									ELSE
										Mach_Control.WJ_b.Error[7]:=TRUE;//尾卷下料时卷针旋转不满足下料角度----20240116
									END_IF	
				     END_IF	
			(*	279:
					IF arrAxisCtrl[AxiseNo.AxisName.TailCurlLine].Cmd.arrbRealPoint[4] THEN
						arrAxisCtrl[AxiseNo.AxisName.TailCurlLine].Cmd.iGoSetPos:=0;
							IF Mach_Control.WJ_b.SinStepMode THEN//尾卷单步模式
								TailCurlSinStep:=TRUE;
							ELSE
								TailCurlSinStep:=FALSE;
							END_IF											
									TailCurlStep3:=280;
					ELSE
						arrAxisCtrl[AxiseNo.AxisName.TailCurlLine].Cmd.iGoSetPos:=4;//尾卷夹电芯平移至取电芯位
					END_IF*)
				
				280://尾卷取电芯夹爪气缸平夹紧
						IF NOT TailCurlSinStep THEN				
							arrCyCtrl[arrCyNo.CylinderName.TailCurlSplintCy].Cmd.bON:=TRUE;//尾卷取料夹爪气缸夹紧
							IF arrCyCtrl[arrCyNo.CylinderName.TailCurlSplintCy].Io.DIOnSwitch THEN
								arrCyCtrl[arrCyNo.ElectValveName.WJ_blow].Cmd.bON:=TRUE;//	夹膜电芯吹气开
								IF Mach_Control.WJ_b.SinStepMode THEN//尾卷单步模式
									TailCurlSinStep:=TRUE;
								ELSE
									TailCurlSinStep:=FALSE;
								END_IF	
								TailCurlStep3:=283;
							END_IF
						END_IF
				
				283://夹膜打开
						IF NOT TailCurlSinStep THEN				
							arrCyCtrl[arrCyNo.CylinderName.PoleSplintCy_D].Cmd.bOFF:=TRUE;
							
							IF arrCyCtrl[arrCyNo.CylinderName.PoleSplintCy_D].Status.OFFState THEN
								IF Mach_Control.WJ_b.SinStepMode THEN//尾卷单步模式
									TailCurlSinStep:=TRUE;
								ELSE
									TailCurlSinStep:=FALSE;
								END_IF
								//arrCyCtrl[arrCyNo.ElectValveName.WJ_blow].Cmd.bON:=FALSE;//	夹膜电芯吹气关
								//arrCyCtrl[arrCyNo.ElectValveName.WJ_blow].Cmd.bOFF:=TRUE;//	夹膜电芯吹气关										
								TailCurlStep3:=287;
							END_IF
						END_IF
					
				287:	
					IF arrCyCtrl[arrCyNo.CylinderName.PoleSplintCy_D].Status.OFFState AND NOT arrAxisCtrl[AxiseNo.AxisName.TailCurlSEPTALine].Status.Coupled AND 
							NOT arrAxisCtrl[AxiseNo.AxisName.TailCurlSEPTAUpDown].Status.Coupled THEN
						IF 	 arrAxis[AxiseNo.AxisName.TailCurlSEPTALine].Status.Homed AND arrAxisCtrl[AxiseNo.AxisName.TailCurlSEPTALine].Status.NoMoving THEN
							IF arrAxisCtrl[AxiseNo.AxisName.TailCurlSEPTALine].Cmd.arrbRealPoint[1] THEN
								arrAxisCtrl[AxiseNo.AxisName.TailCurlSEPTALine].Cmd.iGoSetPos:=0;
							ELSE
								arrAxisCtrl[AxiseNo.AxisName.TailCurlSEPTALine].Cmd.iGoSetPos:=1;//尾卷夹隔膜平移初始位
							END_IF
						END_IF	
						IF 	 arrAxisCtrl[AxiseNo.AxisName.TailCurlSEPTAUpDown].Status.Homed AND arrAxisCtrl[AxiseNo.AxisName.TailCurlSEPTAUpDown].Status.NoMoving THEN
							IF arrAxisCtrl[AxiseNo.AxisName.TailCurlSEPTAUpDown].Cmd.arrbRealPoint[1] THEN
								arrAxisCtrl[AxiseNo.AxisName.TailCurlSEPTAUpDown].Cmd.iGoSetPos:=0;
							ELSE
								arrAxisCtrl[AxiseNo.AxisName.TailCurlSEPTAUpDown].Cmd.iGoSetPos:=1;//尾卷夹隔膜升降初始位
							END_IF
						END_IF
						IF 	arrAxisCtrl[AxiseNo.AxisName.TailCurlSEPTALine].Cmd.arrbRealPoint[1] AND  arrAxisCtrl[AxiseNo.AxisName.TailCurlSEPTAUpDown].Cmd.arrbRealPoint[1]  THEN
								IF Mach_Control.WJ_b.SinStepMode THEN//尾卷单步模式
									TailCurlSinStep:=TRUE;
								ELSE
									TailCurlSinStep:=FALSE;
								END_IF				
								TailCurlStep3:=290;	
						END_IF	
					END_IF			








					290://尾卷压轮升降气缸收回、平移气缸收回
						IF NOT TailCurlSinStep THEN		
								arrCyCtrl[arrCyNo.CylinderName.TailCurlUpdownCy].Cmd.bOFF:=TRUE;//尾卷压轮升降气缸收回
								IF arrCyCtrl[arrCyNo.CylinderName.TailCurlUpdownCy].Io.DIOFFSwitch THEN
									arrCyCtrl[arrCyNo.CylinderName.TailCurlLineCy].Cmd.bOFF:=TRUE;//尾卷压轮平移气缸收回		
									IF arrCyCtrl[arrCyNo.CylinderName.TailCurlLineCy].Io.DIOFFSwitch THEN
										IF Mach_Control.WJ_b.SinStepMode THEN//尾卷单步模式
											TailCurlSinStep:=TRUE;
										ELSE
											TailCurlSinStep:=FALSE;
										END_IF	
										TailCurlStep3:=300;
									END_IF
								END_IF
						END_IF
				300://长、短卷针夹电芯气缸泄压、长、短卷针伸缩轴移动至初始位
						IF NOT TailCurlSinStep THEN			
									IF NOT TON_TailCurl[3].Q THEN
										arrCyCtrl[arrCyNo.CylinderName.CurlingSplintCy_L].Cmd.bFree:=TRUE;//尾卷长卷针泄压
										arrCyCtrl[arrCyNo.CylinderName.CurlingSplintCy_S].Cmd.bFree:=TRUE;//尾卷短卷针泄压
										//arrCyCtrl[arrCyNo.ElectValveName.WJShortvacuum].Cmd.bON:=TRUE;//短卷针张开真空开
										//arrCyCtrl[arrCyNo.CylinderName.CurlingSplintCy_S_1].Cmd.bOFF:=TRUE;//尾卷短卷针泄压
										TON_TailCurl[3].IN:=TRUE;
									ELSE
										IF 	arrAxisCtrl[AxiseNo.AxisName.LCurlingneedleLine].Status.Homed AND arrAxisCtrl[AxiseNo.AxisName.LCurlingneedleLine].Status.NoMoving THEN
											IF arrAxisCtrl[AxiseNo.AxisName.LCurlingneedleLine].Cmd.arrbRealPoint[1] THEN
												arrAxisCtrl[AxiseNo.AxisName.LCurlingneedleLine].Cmd.iGoSetPos:=0;
											ELSE
												arrAxisCtrl[AxiseNo.AxisName.LCurlingneedleLine].Cmd.iGoSetPos:=1;
											END_IF
										END_IF
										IF 	arrAxisCtrl[AxiseNo.AxisName.SCurlingneedleLine].Status.Homed AND arrAxisCtrl[AxiseNo.AxisName.SCurlingneedleLine].Status.NoMoving THEN
											IF arrAxisCtrl[AxiseNo.AxisName.SCurlingneedleLine].Cmd.arrbRealPoint[1] THEN
												arrAxisCtrl[AxiseNo.AxisName.SCurlingneedleLine].Cmd.iGoSetPos:=0;
											ELSE
												arrAxisCtrl[AxiseNo.AxisName.SCurlingneedleLine].Cmd.iGoSetPos:=1;
											END_IF
										END_IF
										IF  arrAxisCtrl[AxiseNo.AxisName.LCurlingneedleLine].Cmd.arrbRealPoint[1] AND arrAxisCtrl[AxiseNo.AxisName.SCurlingneedleLine].Cmd.arrbRealPoint[1] THEN
											TON_TailCurl[3].IN:=FALSE;
											arrCyCtrl[arrCyNo.ElectValveName.WJShortvacuum].Cmd.bON:=TRUE;//短卷针张开真空开
											IF Mach_Control.WJ_b.SinStepMode THEN//尾卷单步模式
												TailCurlSinStep:=TRUE;
											ELSE
												TailCurlSinStep:=FALSE;
											END_IF												
											TailCurlStep3:=305;
										END_IF			
									END_IF
							END_IF	
							
				
							
							
							
							
							
							
							
							
							
				310://尾卷夹电芯平移至初始位
						IF NOT TailCurlSinStep THEN				
								IF 	arrCyCtrl[arrCyNo.CylinderName.TailCurlSplintCy].Io.DIOnSwitch AND  arrAxisCtrl[AxiseNo.AxisName.TailCurlLine].Status.Homed AND arrAxisCtrl[AxiseNo.AxisName.TailCurlLine].Status.NoMoving AND
                                         arrAxisCtrl[AxiseNo.AxisName.LCurlingneedleLine].Cmd.arrbRealPoint[1]  AND arrAxisCtrl[AxiseNo.AxisName.SCurlingneedleLine].Cmd.arrbRealPoint[1]  THEN
									IF arrAxisCtrl[AxiseNo.AxisName.TailCurlLine].Cmd.arrbRealPoint[1] THEN
										arrAxisCtrl[AxiseNo.AxisName.TailCurlLine].Cmd.iGoSetPos:=0;
											IF Mach_Control.WJ_b.SinStepMode THEN//尾卷单步模式
												TailCurlSinStep:=TRUE;
											ELSE
												TailCurlSinStep:=FALSE;
											END_IF										
										TailCurlStep3:=315;
									ELSE
										arrAxisCtrl[AxiseNo.AxisName.TailCurlLine].Cmd.iGoSetPos:=1;//尾卷夹电芯平移至初始位
									END_IF
								END_IF
						END_IF
				
					
						
						315://尾卷夹电芯升降至下电芯位      
						  IF NOT TailCurlSinStep THEN		                                                                                                                                                                                                                                                                                                                                                                                                   		
									IF arrAxisCtrl[AxiseNo.AxisName.TailCurlUpDown].Status.Homed AND arrAxisCtrl[AxiseNo.AxisName.TailCurlUpDown].Status.NoMoving THEN
										IF arrAxisCtrl[AxiseNo.AxisName.TailCurlUpDown].Cmd.arrbRealPoint[3] THEN
											arrAxisCtrl[AxiseNo.AxisName.TailCurlUpDown].Cmd.iGoSetPos:=0;
											IF Mach_Control.WJ_b.SinStepMode THEN//尾卷单步模式
												TailCurlSinStep:=TRUE;
											ELSE
												TailCurlSinStep:=FALSE;
											END_IF									
											TailCurlStep3:=320;
										ELSE
											arrAxisCtrl[AxiseNo.AxisName.TailCurlUpDown].Cmd.iGoSetPos:=3;//尾卷夹电芯升降至下电芯位
										END_IF
									END_IF
							END_IF	
						
						
						
						
				320://尾卷夹电芯旋转至下电芯位
						IF NOT TailCurlSinStep THEN				
								IF 	arrCyCtrl[arrCyNo.CylinderName.TailCurlSplintCy].Status.ONState AND  arrAxisCtrl[AxiseNo.AxisName.TailCurlLine].Status.Homed 
									AND arrAxisCtrl[AxiseNo.AxisName.TailCurlLine].Status.NoMoving AND arrAxisCtrl[AxiseNo.AxisName.GluingLine].Status.Homed AND
									arrAxisCtrl[AxiseNo.AxisName.GluingLine].Status.fActPos<=arrAxispar[AxiseNo.AxisName.GluingLine].arrTargetPoint[10] 
									AND NOT Mach_Control.TJ_b.StickerFlag  THEN
									IF arrAxisCtrl[AxiseNo.AxisName.TailCurlWhirling].Cmd.arrbRealPoint[2] THEN
										arrAxisCtrl[AxiseNo.AxisName.TailCurlWhirling].Cmd.iGoSetPos:=0;
											IF Mach_Control.WJ_b.SinStepMode THEN//尾卷单步模式
												TailCurlSinStep:=TRUE;
											ELSE
												TailCurlSinStep:=FALSE;
											END_IF										
										TailCurlStep3:=325;
									ELSE
										arrAxisCtrl[AxiseNo.AxisName.TailCurlWhirling].Cmd.iGoSetPos:=2;//尾卷夹电芯平移至下电芯位
									END_IF
								END_IF
						END_IF		
						
				
						
			
				325:
				//尾卷夹电芯去避让位   
					(*	  IF NOT TailCurlSinStep THEN		                                                                                                                                                                                                                                                                                                                                                                                                   		
									IF arrAxisCtrl[AxiseNo.AxisName.TailCurlLine].Status.Homed AND arrAxisCtrl[AxiseNo.AxisName.TailCurlLine].Status.NoMoving THEN
										IF arrAxisCtrl[AxiseNo.AxisName.TailCurlLine].Cmd.arrbRealPoint[5] THEN
											arrAxisCtrl[AxiseNo.AxisName.TailCurlLine].Cmd.iGoSetPos:=0;
											IF Mach_Control.WJ_b.SinStepMode THEN//尾卷单步模式
												TailCurlSinStep:=TRUE;
											ELSE
												TailCurlSinStep:=FALSE;
											END_IF									
											TailCurlStep3:=330;
										ELSE
											arrAxisCtrl[AxiseNo.AxisName.TailCurlLine].Cmd.iGoSetPos:=5;//尾卷夹电芯平移至避让位
										END_IF
									END_IF
							END_IF*)
				//尾卷夹电芯去下料避让位
							IF NOT TailCurlSinStep THEN		                                                                                                                                                                                                                                                                                                                                                                                                   		
									IF arrAxisCtrl[AxiseNo.AxisName.TailCurlLine].Status.Homed AND arrAxisCtrl[AxiseNo.AxisName.TailCurlLine].Status.NoMoving THEN
										IF arrAxisCtrl[AxiseNo.AxisName.TailCurlLine].Cmd.arrbRealPoint[10] THEN
											arrAxisCtrl[AxiseNo.AxisName.TailCurlLine].Cmd.iGoSetPos:=0;
											IF Mach_Control.WJ_b.SinStepMode THEN//尾卷单步模式
												TailCurlSinStep:=TRUE;
											ELSE
												TailCurlSinStep:=FALSE;
											END_IF									
											TailCurlStep3:=330;
										ELSE
											arrAxisCtrl[AxiseNo.AxisName.TailCurlLine].Cmd.iGoSetPos:=10;//尾卷夹电芯平移至避让位
										END_IF
									END_IF
							END_IF
				330:
						IF NOT TailCurlSinStep THEN
								Mach_Control.WJ_b.TailCultOffloading:=TRUE;//下电芯请求														
								TailCurlStep3:=332;
								
								IF Mach_Control.WJ_b.SinStepMode THEN//尾卷单步模式
									TailCurlSinStep:=TRUE;
								ELSE
									TailCurlSinStep:=FALSE;
								END_IF					
						END_IF				
						

				332:   ///////////////////
						
					IF 	arrAxisCtrl[AxiseNo.AxisName.GluingLine].Cmd.arrbRealPoint[8] AND arrAxisCtrl[AxiseNo.AxisName.GluingLine].Status.NoMoving
						AND arrAxisCtrl[AxiseNo.AxisName.GluingWhirling].Cmd.arrbRealPoint[5] AND arrAxisCtrl[AxiseNo.AxisName.GluingWhirling].Status.NoMoving
						AND arrCyCtrl[arrCyNo.CylinderName.PullGlueModelCy].Status.ONState AND NOT arrCyCtrl[arrCyNo.CylinderName.PullGlueModelCy].Status.Error2 
						AND arrAxisCtrl[AxiseNo.AxisName.TailCurlLine].Status.Homed AND arrAxisCtrl[AxiseNo.AxisName.TailCurlLine].Status.NoMoving	
						AND NOT Mach_Control.TJ_b.StickerDone  AND NOT Mach_Control.TJ_b.StickerFlag
						AND NOT CellMemory[Mach_Control.TJ_b.TJ_Memory].Cell AND NOT Mach_Control.se.GluebHave	THEN
						TailCurlStep3:=335;

					END_IF
						
				335:
						IF arrAxisCtrl[AxiseNo.AxisName.TailCurlLine].Cmd.arrbRealPoint[6] THEN
							arrAxisCtrl[AxiseNo.AxisName.TailCurlLine].Cmd.iGoSetPos:=0;
							IF Mach_Control.WJ_b.SinStepMode THEN//尾卷单步模式
								TailCurlSinStep:=TRUE;
							ELSE
								TailCurlSinStep:=FALSE;
							END_IF									
							TailCurlStep3:=336;
						ELSE
							arrAxisCtrl[AxiseNo.AxisName.TailCurlLine].Cmd.iGoSetPos:=6;//尾卷夹电芯平移至下电芯位
						END_IF
						
				336:
							IF NOT TailCurlSinStep THEN		
									IF 	arrAxisCtrl[AxiseNo.AxisName.GluingLine].Cmd.arrbRealPoint[8] AND arrAxisCtrl[AxiseNo.AxisName.GluingLine].Status.NoMoving
										AND arrAxisCtrl[AxiseNo.AxisName.GluingWhirling].Cmd.arrbRealPoint[5] AND arrAxisCtrl[AxiseNo.AxisName.GluingWhirling].Status.NoMoving
										AND arrCyCtrl[arrCyNo.CylinderName.PullGlueModelCy].Status.ONState AND NOT arrCyCtrl[arrCyNo.CylinderName.PullGlueModelCy].Status.Error2 
										AND arrAxisCtrl[AxiseNo.AxisName.TailCurlRetracting].Status.Homed AND arrAxisCtrl[AxiseNo.AxisName.TailCurlRetracting].Status.NoMoving		THEN
									IF arrAxisCtrl[AxiseNo.AxisName.TailCurlRetracting].Cmd.arrbRealPoint[3] THEN
										arrAxisCtrl[AxiseNo.AxisName.TailCurlRetracting].Cmd.iGoSetPos:=0;
										IF Mach_Control.WJ_b.SinStepMode THEN//尾卷单步模式
											TailCurlSinStep:=TRUE;
										ELSE
											TailCurlSinStep:=FALSE;
										END_IF									
										TailCurlStep3:=337;
									ELSE
										arrAxisCtrl[AxiseNo.AxisName.TailCurlRetracting].Cmd.iGoSetPos:=3;//尾卷夹电芯伸缩至下电芯位
										END_IF
									END_IF
							END_IF	
				337:
							IF NOT TailCurlSinStep THEN			
								IF 	arrAxisCtrl[AxiseNo.AxisName.TailCurlUpDown].Status.Homed AND arrAxisCtrl[AxiseNo.AxisName.TailCurlUpDown].Status.NoMoving  THEN
									IF arrAxisCtrl[AxiseNo.AxisName.TailCurlUpDown].Cmd.arrbRealPoint[4] THEN
													arrAxisCtrl[AxiseNo.AxisName.TailCurlUpDown].Cmd.iGoSetPos:=0;
													IF Mach_Control.WJ_b.SinStepMode THEN//尾卷单步模式
													TailCurlSinStep:=TRUE;
													ELSE
														TailCurlSinStep:=FALSE;
													END_IF	
													TailCurlStep3:=338;
									ELSE
													arrAxisCtrl[AxiseNo.AxisName.TailCurlUpDown].Cmd.iGoSetPos:=4;//尾卷夹电芯升降至下电芯位
									END_IF
								END_IF	
						END_IF				
						
						
						
						
						
						
				338:
				
						IF NOT TailCurlSinStep THEN				
							arrCyCtrl[arrCyNo.CylinderName.PullGlueModelCy].Cmd.bOFF:=TRUE;//贴胶治具气缸闭合
							IF arrCyCtrl[arrCyNo.CylinderName.PullGlueModelCy].Status.OFFState THEN
								IF Mach_Control.WJ_b.SinStepMode THEN//尾卷单步模式
									TailCurlSinStep:=TRUE;
								ELSE
									TailCurlSinStep:=FALSE;
								END_IF										
								TailCurlStep3:=339;
							END_IF
						END_IF


				339:
				

					IF NOT TailCurlSinStep THEN				
							arrCyCtrl[arrCyNo.CylinderName.TailCurlSplintCy].Cmd.bOFF:=TRUE;//尾卷夹爪气缸打开
							IF arrCyCtrl[arrCyNo.CylinderName.TailCurlSplintCy].Status.OFFState THEN
								arrCyCtrl[arrCyNo.ElectValveName.WJ_blow].Cmd.bOFF:=TRUE;//	夹膜电芯吹气关
								IF Mach_Control.WJ_b.SinStepMode THEN//尾卷单步模式
									TailCurlSinStep:=TRUE;
								ELSE
									TailCurlSinStep:=FALSE;
								END_IF	
								Mach_Control.TJ_b.StickerFlag:=TRUE;//置位贴胶夹爪有料标记
								TailCurlStep3:=340;
							END_IF
						END_IF

				340:
					IF NOT TailCurlSinStep THEN			
						IF 	arrAxisCtrl[AxiseNo.AxisName.TailCurlUpDown].Status.Homed AND arrAxisCtrl[AxiseNo.AxisName.TailCurlUpDown].Status.NoMoving  AND
							arrAxisCtrl[AxiseNo.AxisName.TailCurlUpDown].Cmd.arrbRealPoint[4] THEN
							arrAxisPar[AxiseNo.AxisName.TailCurlUpDown].fVelocity_of_Rel := 20   ;
							arrAxisCtrl[AxiseNo.AxisName.TailCurlUpDown].Cmd.fPosition_of_Rel :=3 ;
							arrAxisCtrl[AxiseNo.AxisName.TailCurlUpDown].Cmd.bMoveRel :=  TRUE ;
						END_IF
							IF arrAxis[AxiseNo.AxisName.TailCurlUpDown].NcToPlc.SetPos-arrAxisPar[AxiseNo.AxisName.TailCurlUpDown].arrTargetPoint[4] >=3  
							AND arrAxisCtrl[AxiseNo.AxisName.TailCurlUpDown].Status.NoMoving THEN
								IF Mach_Control.WJ_b.SinStepMode THEN//尾卷单步模式
									TailCurlSinStep:=TRUE;
								ELSE
									TailCurlSinStep:=FALSE;
								END_IF
								TailCurlStep3:=341;
							END_IF
					END_IF	
							
				341:// 尾卷夹电芯平移至避让位

						IF NOT TailCurlSinStep THEN			
								IF 	arrAxisCtrl[AxiseNo.AxisName.TailCurlLine].Status.Homed AND arrAxisCtrl[AxiseNo.AxisName.TailCurlLine].Status.NoMoving THEN
									IF arrAxisCtrl[AxiseNo.AxisName.TailCurlLine].Cmd.arrbRealPoint[10] THEN
										arrAxisCtrl[AxiseNo.AxisName.TailCurlLine].Cmd.iGoSetPos:=0;
									IF Mach_Control.WJ_b.SinStepMode THEN//尾卷单步模式
									TailCurlSinStep:=TRUE;
								ELSE
									TailCurlSinStep:=FALSE;
								END_IF	
										TailCurlStep3:=343;
									ELSE
										arrAxisCtrl[AxiseNo.AxisName.TailCurlLine].Cmd.iGoSetPos:=10;//尾卷夹电芯平移至避让位
									END_IF
								END_IF	
						END_IF	
				343:	
					CellMemory[Mach_Control.TJ_b.TJ_Memory]:=CellMemory[Mach_Control.WJ_b.WJ_Memory];
					MEMSET(ADR(CellMemory[Mach_Control.WJ_b.WJ_Memory]),0,SIZEOF(CellMemory[Mach_Control.WJ_b.WJ_Memory]));		
					TailCurlStep3:=345;		
						
						
						
						
						
						
						
				345:
		
						IF NOT TailCurlSinStep THEN			
								IF 	arrAxisCtrl[AxiseNo.AxisName.TailCurlRetracting].Status.Homed AND arrAxisCtrl[AxiseNo.AxisName.TailCurlRetracting].Status.NoMoving THEN
									IF arrAxisCtrl[AxiseNo.AxisName.TailCurlRetracting].Cmd.arrbRealPoint[1] THEN
										arrAxisCtrl[AxiseNo.AxisName.TailCurlRetracting].Cmd.iGoSetPos:=0;
										IF Mach_Control.WJ_b.SinStepMode THEN//尾卷单步模式
									TailCurlSinStep:=TRUE;
								ELSE
									TailCurlSinStep:=FALSE;
								END_IF	
										
										TailCurlStep3:=350;
									ELSE
										arrAxisCtrl[AxiseNo.AxisName.TailCurlRetracting].Cmd.iGoSetPos:=1;//尾卷夹电芯伸缩回到初始位
									END_IF
								END_IF	
						END_IF	
						
						
						
						
				350:
				IF NOT TailCurlSinStep THEN		
					 IF arrAxisCtrl[AxiseNo.AxisName.GluingLine].Status.fActPos<=arrAxispar[AxiseNo.AxisName.GluingLine].arrTargetPoint[10] 
						AND arrAxisCtrl[AxiseNo.AxisName.GluingLine].Status.Homed AND NOT Mach_Control.WJ_b.TailCultOffloading AND arrAxisCtrl[AxiseNo.AxisName.TailCurlLine].Status.Homed 
						AND arrAxisCtrl[AxiseNo.AxisName.TailCurlLine].Status.NoMoving THEN
						
								IF arrAxisCtrl[AxiseNo.AxisName.TailCurlLine].Cmd.arrbRealPoint[1] THEN
									IF Mach_Control.WJ_b.SinStepMode THEN//尾卷单步模式
									TailCurlSinStep:=TRUE;
								ELSE
									TailCurlSinStep:=FALSE;
								END_IF	
									arrAxisCtrl[AxiseNo.AxisName.TailCurlLine].Cmd.iGoSetPos:=0;
									
									TailCurlStep3:=355;
								ELSE
									arrAxisCtrl[AxiseNo.AxisName.TailCurlLine].Cmd.iGoSetPos:=1;//尾卷夹电芯平移至初始位
								END_IF
						END_IF	
				END_IF	

				355:
							IF NOT TailCurlSinStep THEN			
								IF 	arrAxisCtrl[AxiseNo.AxisName.TailCurlUpDown].Status.Homed AND arrAxisCtrl[AxiseNo.AxisName.TailCurlUpDown].Status.NoMoving  THEN
									IF arrAxisCtrl[AxiseNo.AxisName.TailCurlUpDown].Cmd.arrbRealPoint[4] THEN
													arrAxisCtrl[AxiseNo.AxisName.TailCurlUpDown].Cmd.iGoSetPos:=0;
													IF Mach_Control.WJ_b.SinStepMode THEN//尾卷单步模式
													TailCurlSinStep:=TRUE;
													ELSE
														TailCurlSinStep:=FALSE;
													END_IF	
													TailCurlStep3:=360;
									ELSE
													arrAxisCtrl[AxiseNo.AxisName.TailCurlUpDown].Cmd.iGoSetPos:=4;//尾卷夹电芯升降至下电芯位
									END_IF
								END_IF	
						END_IF
				360:
					IF NOT TailCurlSinStep THEN		
					 IF arrAxisCtrl[AxiseNo.AxisName.GluingLine].Status.fActPos<=arrAxispar[AxiseNo.AxisName.GluingLine].arrTargetPoint[10] 
						AND arrAxisCtrl[AxiseNo.AxisName.GluingLine].Status.Homed AND NOT Mach_Control.WJ_b.TailCultOffloading AND arrAxis[AxiseNo.AxisName.TailCurlWhirling].Status.Homed 
						AND arrAxisCtrl[AxiseNo.AxisName.TailCurlWhirling].Status.NoMoving AND arrAxisCtrl[AxiseNo.AxisName.TailCurlLine].Status.NoMoving AND arrAxisCtrl[AxiseNo.AxisName.TailCurlLine].Cmd.arrbRealPoint[1] THEN
						
								IF arrAxisCtrl[AxiseNo.AxisName.TailCurlWhirling].Cmd.arrbRealPoint[1] THEN
									IF Mach_Control.WJ_b.SinStepMode THEN//尾卷单步模式
									TailCurlSinStep:=TRUE;
								ELSE
									TailCurlSinStep:=FALSE;
								END_IF	
									arrAxisCtrl[AxiseNo.AxisName.TailCurlWhirling].Cmd.iGoSetPos:=0;
									//Mach_Control.WJ_b.TailCultOffloadingDone:=TRUE;
									TailCurlStep3:=370;
								ELSE
									arrAxisCtrl[AxiseNo.AxisName.TailCurlWhirling].Cmd.iGoSetPos:=1;//尾卷夹电芯旋转至取电芯位
								END_IF
						END_IF	
				END_IF	
                
				 370://尾卷夹电芯平移去取电芯等待位
					 IF NOT TailCurlSinStep THEN	
							 IF  arrAxisCtrl[AxiseNo.AxisName.TailCurlUpDown].Status.Homed AND arrAxisCtrl[AxiseNo.AxisName.TailCurlUpDown].Status.NoMoving THEN
											IF arrAxisCtrl[AxiseNo.AxisName.TailCurlUpDown].Cmd.arrbRealPoint[1] THEN
												arrAxisCtrl[AxiseNo.AxisName.TailCurlUpDown].Cmd.iGoSetPos:=0;
											ELSE
												arrAxisCtrl[AxiseNo.AxisName.TailCurlUpDown].Cmd.iGoSetPos:=1;//尾卷夹升降去取电芯高度
											END_IF
							 END_IF
						 
						   IF arrAxisCtrl[AxiseNo.AxisName.TailCurlWhirling].Cmd.arrbRealPoint[1] AND arrAxisCtrl[AxiseNo.AxisName.TailCurlUpDown].Cmd.arrbRealPoint[1] AND
							  arrAxisCtrl[AxiseNo.AxisName.TailCurlSEPTALine].Cmd.arrbRealPoint[1] AND  arrAxisCtrl[AxiseNo.AxisName.TailCurlSEPTAUpDown].Cmd.arrbRealPoint[1] AND
							  arrAxisCtrl[AxiseNo.AxisName.LCurlingneedleLine].Cmd.arrbRealPoint[1] AND arrAxisCtrl[AxiseNo.AxisName.SCurlingneedleLine].Cmd.arrbRealPoint[1] AND
							  arrCyCtrl[arrCyNo.CylinderName.PoleSplintCy_D].Io.DIOFFSwitch AND arrCyCtrl[arrCyNo.CylinderName.TailCurlUpdownCy].Io.DIOFFSwitch AND
							  arrAxisCtrl[AxiseNo.AxisName.TailCurlLine].Status.Homed AND arrAxisCtrl[AxiseNo.AxisName.TailCurlLine].Status.NoMoving  THEN
								   IF arrAxisCtrl[AxiseNo.AxisName.TailCurlLine].Cmd.arrbRealPoint[11]  THEN
									  arrAxisCtrl[AxiseNo.AxisName.TailCurlLine].Cmd.iGoSetPos:=0;
										IF Mach_Control.WJ_b.SinStepMode THEN//尾卷单步模式
										   TailCurlSinStep:=TRUE;
										ELSE
										   TailCurlSinStep:=FALSE;
										END_IF									
										   TailCurlStep3:=0;
										   TailCurlTorMark:=FALSE;//尾卷夹电芯平移力矩判断标志位
								   ELSE
									   arrAxisCtrl[AxiseNo.AxisName.TailCurlLine].Cmd.iGoSetPos:=11;//尾卷夹电芯平移去取电芯等待位
									   TailCurlTorMark:=TRUE;//尾卷夹电芯平移力矩判断标志位
								   END_IF   
							END_IF
						END_IF
				//////////////////////////////////////////////////////////////////////////////////////
				///////////////////////////////////叠台空叠隔膜不尾卷/////////////////////////////////////////////////////
				900:
					    IF NOT TailCurlSinStep THEN
							IF  Mach_Control.DT_b.OffloadRequest AND DP_Step0=6040  THEN
								IF 	arrAxisCtrl[AxiseNo.AxisName.TailCurlUpDown].Status.Homed AND arrAxisCtrl[AxiseNo.AxisName.TailCurlUpDown].Status.NoMoving THEN
										IF arrAxisCtrl[AxiseNo.AxisName.TailCurlUpDown].Cmd.arrbRealPoint[1] THEN//尾卷夹电芯升降初始位
											arrAxisCtrl[AxiseNo.AxisName.TailCurlUpDown].Cmd.iGoSetPos:=0;
										ELSE
											arrAxisCtrl[AxiseNo.AxisName.TailCurlUpDown].Cmd.iGoSetPos:=1;
										END_IF
									END_IF	
								IF 	arrAxisCtrl[AxiseNo.AxisName.TailCurlSEPTAUpDown].Status.Homed AND arrAxisCtrl[AxiseNo.AxisName.TailCurlSEPTAUpDown].Status.NoMoving THEN
										IF arrAxisCtrl[AxiseNo.AxisName.TailCurlSEPTAUpDown].Cmd.arrbRealPoint[1] THEN//夹膜升降初始位
											arrAxisCtrl[AxiseNo.AxisName.TailCurlSEPTAUpDown].Cmd.iGoSetPos:=0;
										ELSE
											arrAxisCtrl[AxiseNo.AxisName.TailCurlSEPTAUpDown].Cmd.iGoSetPos:=1;
										END_IF
									END_IF	
									IF 	arrAxisCtrl[AxiseNo.AxisName.TailCurlUpDown].Cmd.arrbRealPoint[1]  AND arrAxisCtrl[AxiseNo.AxisName.TailCurlUpDown].Cmd.arrbRealPoint[1] 
										AND arrAxisCtrl[AxiseNo.AxisName.TailCurlSEPTAUpDown].Cmd.arrbRealPoint[1]  AND arrAxisCtrl[AxiseNo.AxisName.TailCurlSEPTAUpDown].Cmd.arrbRealPoint[1]	THEN
										IF Mach_Control.WJ_b.SinStepMode THEN//尾卷单步模式
											TailCurlSinStep:=TRUE;
										ELSE
											TailCurlSinStep:=FALSE;
										END_IF								
										TailCurlStep3:=1010;	
										TON_TailCurl[6].IN:=FALSE;
									END_IF
							ELSE
								TailCurlStep3:=0;
							END_IF	
					END_IF
					
				
				
				
				/////////////////////////////////////////////////////////////////////////////////////////////////////
				/////////////////////////////////////////////////////////////////////////////////////////////////////////
				(*1000:
					Par.stDT_date.BH_Thickness :=((Par.stDT_date.An_Thickness+Par.stDT_date.SEPTA_Thickness)*Par.stDT_date.An_Quantity+(Par.stDT_date.Ca_Thickness+Par.stDT_date.SEPTA_Thickness)*Par.stDT_date.Ca_Quantity)-((Par.stDT_date.An_Thickness+Par.stDT_date.SEPTA_Thickness)*Mach_Control.An_b.An_Quantited+(Par.stDT_date.Ca_Thickness+Par.stDT_date.SEPTA_Thickness)*Mach_Control.Ca_b.Ca_Quantited);
					TailCurlStep3:=1001;

				1001:
					arrAxispar[AxiseNo.AxisName.TailCurlUpDown].arrTargetPoint[6]:=arrAxispar[AxiseNo.AxisName.TailCurlUpDown].arrTargetPoint[1]-Par.stDT_date.BH_Thickness;
					arrAxispar[AxiseNo.AxisName.TailCurlSEPTAUpDown].arrTargetPoint[3]:=arrAxispar[AxiseNo.AxisName.TailCurlSEPTAUpDown].arrTargetPoint[1]+Par.stDT_date.BH_Thickness;
					TailCurlStep3:=1005;*)




				1000://夹膜升降去取电芯位，夹电芯升降去取电芯位	
						
					    IF NOT TailCurlSinStep THEN
							IF  Mach_Control.DT_b.OffloadRequest THEN
								IF 	arrAxisCtrl[AxiseNo.AxisName.TailCurlUpDown].Status.Homed AND arrAxisCtrl[AxiseNo.AxisName.TailCurlUpDown].Status.NoMoving THEN
										IF arrAxisCtrl[AxiseNo.AxisName.TailCurlUpDown].Cmd.arrbRealPoint[6] THEN
											arrAxisCtrl[AxiseNo.AxisName.TailCurlUpDown].Cmd.iGoSetPos:=0;
										ELSE
											arrAxisCtrl[AxiseNo.AxisName.TailCurlUpDown].Cmd.iGoSetPos:=6;
										END_IF
									END_IF	
								IF 	arrAxisCtrl[AxiseNo.AxisName.TailCurlSEPTAUpDown].Status.Homed AND arrAxisCtrl[AxiseNo.AxisName.TailCurlSEPTAUpDown].Status.NoMoving THEN
										IF arrAxisCtrl[AxiseNo.AxisName.TailCurlSEPTAUpDown].Cmd.arrbRealPoint[3] THEN
											arrAxisCtrl[AxiseNo.AxisName.TailCurlSEPTAUpDown].Cmd.iGoSetPos:=0;
										ELSE
											arrAxisCtrl[AxiseNo.AxisName.TailCurlSEPTAUpDown].Cmd.iGoSetPos:=3;
										END_IF
									END_IF	
									IF 	arrAxisCtrl[AxiseNo.AxisName.TailCurlUpDown].Cmd.arrbRealPoint[6]  AND arrAxisCtrl[AxiseNo.AxisName.TailCurlUpDown].Status.NoMoving
										AND arrAxisCtrl[AxiseNo.AxisName.TailCurlSEPTAUpDown].Cmd.arrbRealPoint[3]  AND arrAxisCtrl[AxiseNo.AxisName.TailCurlSEPTAUpDown].Status.NoMoving	THEN
										IF Mach_Control.WJ_b.SinStepMode THEN//尾卷单步模式
											TailCurlSinStep:=TRUE;
										ELSE
											TailCurlSinStep:=FALSE;
										END_IF								
										TailCurlStep3:=1010;	
									END_IF
								ELSE
								TailCurlStep3:=0;
								END_IF	
					END_IF
					
		
					
				1010://负极叠片搬运平移轴在安全位置，尾卷夹电芯平移至取电芯位 、尾卷夹电芯伸缩至取电芯位 、尾卷夹膜平移至隔膜切断位///////////////////
	                 IF    NOT TailCurlSinStep AND  arrAxisCtrl[AxiseNo.AxisName.TailCurlLine].Status.Homed AND arrAxisCtrl[AxiseNo.AxisName.TailCurlLine].Status.NoMoving AND  
                           arrAxisCtrl[AxiseNo.AxisName.CaDTCarryingLine].Cmd.arrbRealPoint[1] AND arrAxisCtrl[AxiseNo.AxisName.CaDTCarryingUpDown].Cmd.arrbRealPoint[5] AND
                             arrAxisCtrl[AxiseNo.AxisName.TailCurlWhirling].Cmd.arrbRealPoint[1] AND arrAxisCtrl[AxiseNo.AxisName.SEPTATLine].Cmd.arrbRealPoint[1] AND
							 arrAxisCtrl[AxiseNo.AxisName.TailCurlSEPTAUpDown].Cmd.arrbRealPoint[3] AND arrAxisCtrl[AxiseNo.AxisName.TailCurlUpDown].Cmd.arrbRealPoint[6] AND
							  arrAxisCtrl[AxiseNo.AxisName.LCurlingneedleLine].Cmd.arrbRealPoint[1]  AND arrAxisCtrl[AxiseNo.AxisName.SCurlingneedleLine].Cmd.arrbRealPoint[1]   AND
							arrCyCtrl[arrCyNo.CylinderName.TailCurlSplintCy].Status.OFFState AND arrCyCtrl[arrCyNo.CylinderName.PoleSplintCy_D].Status.OFFState  AND
                            arrCyCtrl[arrCyNo.CylinderName.PoleHotCutterCy].Status.OFFState   THEN			
			
									IF 	 Mach_Control.DT_b.OffloadRequest THEN	
										TailCurlStep3:=1016;		
										(*	
											arrAxisCtrl[AxiseNo.AxisName.TailCurlSEPTALine].Cmd.fOverride:=100;
											arrAxisCtrl[AxiseNo.AxisName.TailCurlRetracting].Cmd.fOverride:=100;
											arrAxisCtrl[AxiseNo.AxisName.TailCurlLine].Cmd.fOverride:=100;
											
											IF   arrAxis[AxiseNo.AxisName.TailCurlSEPTALine].Status.Homed AND arrAxisCtrl[AxiseNo.AxisName.TailCurlSEPTALine].Status.NoMoving THEN
												IF arrAxisCtrl[AxiseNo.AxisName.TailCurlSEPTALine].Cmd.arrbRealPoint[2] THEN
													arrAxisCtrl[AxiseNo.AxisName.TailCurlSEPTALine].Cmd.iGoSetPos:=0;
												ELSE
													arrAxisCtrl[AxiseNo.AxisName.TailCurlSEPTALine].Cmd.iGoSetPos:=2;//尾卷夹隔膜平移取芯位
												END_IF
											END_IF
											IF 	arrAxisCtrl[AxiseNo.AxisName.TailCurlRetracting].Status.Homed AND arrAxisCtrl[AxiseNo.AxisName.TailCurlRetracting].Status.NoMoving THEN
												IF arrAxisCtrl[AxiseNo.AxisName.TailCurlRetracting].Cmd.arrbRealPoint[2] THEN
													arrAxisCtrl[AxiseNo.AxisName.TailCurlRetracting].Cmd.iGoSetPos:=0;
												ELSE
													arrAxisCtrl[AxiseNo.AxisName.TailCurlRetracting].Cmd.iGoSetPos:=2;//尾卷夹电芯伸缩至取电芯位
												END_IF
											END_IF					
											IF 	arrAxisCtrl[AxiseNo.AxisName.TailCurlLine].Status.Homed AND arrAxisCtrl[AxiseNo.AxisName.TailCurlLine].Status.NoMoving THEN
												IF arrAxisCtrl[AxiseNo.AxisName.TailCurlLine].Cmd.arrbRealPoint[2] THEN
													arrAxisCtrl[AxiseNo.AxisName.TailCurlLine].Cmd.iGoSetPos:=0;
												ELSE
													arrAxisCtrl[AxiseNo.AxisName.TailCurlLine].Cmd.iGoSetPos:=2;//尾卷夹电芯平移至取电芯位
												END_IF
											END_IF						
											IF arrAxisCtrl[AxiseNo.AxisName.TailCurlSEPTALine].Cmd.arrbRealPoint[2] AND arrAxisCtrl[AxiseNo.AxisName.TailCurlRetracting].Cmd.arrbRealPoint[2] AND
												arrAxisCtrl[AxiseNo.AxisName.TailCurlLine].Cmd.arrbRealPoint[2]  THEN
												IF  Mach_Control.WJ_b.SinStepMode THEN//尾卷单步模式
													TailCurlSinStep:=TRUE;
												ELSE
													TailCurlSinStep:=FALSE;
												END_IF	
												TailCurlStep3:=1020;
												TailCurlSplintCy_TON.IN:=FALSE;	
											END_IF
										*)
									ELSE
										TailCurlStep3:=0;
									END_IF	
						ELSE
										Mach_Control.WJ_b.Error[11]:=TRUE;	//尾卷夹电芯平移至取电芯位时条件不满足报警									
						END_IF	

				1016:
					tailCurlGearInEnable1:=TRUE;//夹电芯平移与夹膜平移电子齿轮----取料
					tailRetGearInEnable:=TRUE;//夹电芯平移与夹电芯伸缩电子齿轮
					IF tailCurl_GearIn1.InGear AND tailRetGearIn.InGear THEN
						TailCurlStep3:=1017;
					END_IF			
				1017:
					IF 	arrAxisCtrl[AxiseNo.AxisName.TailCurlLine].Status.Homed AND 
                           arrAxisCtrl[AxiseNo.AxisName.CaDTCarryingLine].Cmd.arrbRealPoint[1] AND arrAxisCtrl[AxiseNo.AxisName.CaDTCarryingUpDown].Cmd.arrbRealPoint[5] AND
                             arrAxisCtrl[AxiseNo.AxisName.TailCurlWhirling].Cmd.arrbRealPoint[1] AND arrAxisCtrl[AxiseNo.AxisName.SEPTATLine].Cmd.arrbRealPoint[1] AND
							 arrAxisCtrl[AxiseNo.AxisName.TailCurlSEPTAUpDown].Cmd.arrbRealPoint[3] AND arrAxisCtrl[AxiseNo.AxisName.TailCurlUpDown].Cmd.arrbRealPoint[6] AND
							  arrAxisCtrl[AxiseNo.AxisName.LCurlingneedleLine].Cmd.arrbRealPoint[1]  AND arrAxisCtrl[AxiseNo.AxisName.SCurlingneedleLine].Cmd.arrbRealPoint[1]   AND
							arrCyCtrl[arrCyNo.CylinderName.TailCurlSplintCy].Status.OFFState AND arrCyCtrl[arrCyNo.CylinderName.PoleSplintCy_D].Status.OFFState  AND
                            arrCyCtrl[arrCyNo.CylinderName.PoleHotCutterCy].Status.OFFState       THEN
									IF arrAxisCtrl[AxiseNo.AxisName.TailCurlLine].Cmd.arrbRealPoint[2] AND arrAxisCtrl[AxiseNo.AxisName.TailCurlLine].Status.NoMoving THEN
										TailCurlTorMark:=FALSE;//尾卷夹电芯平移力矩判断标志位
										arrAxisCtrl[AxiseNo.AxisName.TailCurlLine].Cmd.iGoSetPos:=0;
										TailCurlStep3:=1018;
									ELSE
										arrAxisCtrl[AxiseNo.AxisName.TailCurlLine].Cmd.iGoSetPos:=2;//尾卷夹电芯平移至取电芯位
										TailCurlTorMark:=TRUE;//尾卷夹电芯平移力矩判断标志位
									END_IF
					ELSE
										Mach_Control.WJ_b.Error[11]:=TRUE;	//尾卷夹电芯平移至取电芯位时条件不满足报警
					END_IF		
				1018:
					IF arrAxisCtrl[AxiseNo.AxisName.TailCurlSEPTALine].Cmd.arrbRealPoint[2] AND arrAxisCtrl[AxiseNo.AxisName.TailCurlRetracting].Cmd.arrbRealPoint[2] AND
						arrAxisCtrl[AxiseNo.AxisName.TailCurlLine].Cmd.arrbRealPoint[2]  THEN
						tailCurlGearInEnable1:=FALSE;//夹电芯平移与夹膜平移电子齿轮----取料
						tailRetGearInEnable:=FALSE;//夹电芯平移与夹电芯伸缩电子齿轮
					END_IF
					IF NOT tailCurl_GearIn1.InGear AND NOT tailRetGearIn.InGear THEN
						TailCurlStep3:=1020;
					END_IF			




				
				1020://尾卷夹电芯气缸夹紧//////////////////////////////
						arrAxisCtrl[AxiseNo.AxisName.TailCurlSEPTALine].Cmd.fOverride:=100;
						arrAxisCtrl[AxiseNo.AxisName.TailCurlRetracting].Cmd.fOverride:=100;
						arrAxisCtrl[AxiseNo.AxisName.TailCurlLine].Cmd.fOverride:=100;
						IF NOT TailCurlSinStep THEN					
							arrCyCtrl[arrCyNo.CylinderName.TailCurlSplintCy].Cmd.bON:=TRUE;//尾卷取料夹爪气缸夹紧
							TailCurlSplintCy_TON.IN:=TRUE;					
							IF (*arrCyCtrl[arrCyNo.CylinderName.TailCurlSplintCy].Io.DIOnSwitch OR*) TailCurlSplintCy_TON.Q THEN
								IF Mach_Control.WJ_b.SinStepMode THEN//尾卷单步模式
									TailCurlSinStep:=TRUE;
								ELSE
									TailCurlSinStep:=FALSE;
								END_IF								
								TailCurlStep3:=1030;
								Mach_Control.DT_b.OffloadRequest:=FALSE;//复位电芯下料请求
								TailCurlSplintCy_TON.IN:=FALSE;	
							END_IF
						END_IF
				1030://叠台升降下降至下电芯位	
					IF NOT TailCurlSinStep THEN				
								IF 	arrAxisCtrl[AxiseNo.AxisName.DTUpDown].Status.Homed   THEN
										arrAxisCtrl[AxiseNo.AxisName.DTUpDown].Cmd.bHome:=FALSE;//叠台升降下降至下电芯位回原点
												IF arrAxisCtrl[AxiseNo.AxisName.DTUpDown].Status.NoMoving THEN
															IF arrAxisCtrl[AxiseNo.AxisName.DTUpDown].Cmd.arrbRealPoint[2] THEN
																arrAxisCtrl[AxiseNo.AxisName.DTUpDown].Cmd.iGoSetPos:=0;
																IF Mach_Control.WJ_b.SinStepMode THEN//尾卷单步模式
																	TailCurlSinStep:=TRUE;
																ELSE
																	TailCurlSinStep:=FALSE;
																END_IF									
																TailCurlStep3:=1040;
															ELSE
																arrAxisCtrl[AxiseNo.AxisName.DTUpDown].Cmd.iGoSetPos:=2;//叠台升降下降至下电芯位
															END_IF
											END_IF
								ELSE
										arrAxisCtrl[AxiseNo.AxisName.DTUpDown].Cmd.bHome:=TRUE;//叠台升降下降至下电芯位回原点
								END_IF	
					END_IF
				1040://左、右压刀升降轴上升至抽刀高度
						IF NOT TailCurlSinStep THEN						
								IF 	arrAxisCtrl[AxiseNo.AxisName.LeftYDUpDown].Status.Homed AND arrAxisCtrl[AxiseNo.AxisName.LeftYDUpDown].Status.NoMoving THEN
									IF arrAxisCtrl[AxiseNo.AxisName.LeftYDUpDown].Cmd.arrbRealPoint[4] THEN
										arrAxisCtrl[AxiseNo.AxisName.LeftYDUpDown].Cmd.iGoSetPos:=0;
									ELSE
										arrAxisCtrl[AxiseNo.AxisName.LeftYDUpDown].Cmd.iGoSetPos:=4;//左压刀升降轴上升至抽刀高度
									END_IF
								END_IF					
								IF 	arrAxisCtrl[AxiseNo.AxisName.RightYDUpDown].Status.Homed AND arrAxisCtrl[AxiseNo.AxisName.RightYDUpDown].Status.NoMoving THEN
									IF arrAxisCtrl[AxiseNo.AxisName.RightYDUpDown].Cmd.arrbRealPoint[4] THEN
										arrAxisCtrl[AxiseNo.AxisName.RightYDUpDown].Cmd.iGoSetPos:=0;
									ELSE
										arrAxisCtrl[AxiseNo.AxisName.RightYDUpDown].Cmd.iGoSetPos:=4;//右压好升降上升至抽刀高度
									END_IF
								END_IF				
								IF arrAxisCtrl[AxiseNo.AxisName.LeftYDUpDown].Cmd.arrbRealPoint[4] AND arrAxisCtrl[AxiseNo.AxisName.RightYDUpDown].Cmd.arrbRealPoint[4] THEN
									IF Mach_Control.WJ_b.SinStepMode THEN//尾卷单步模式
										TailCurlSinStep:=TRUE;
									ELSE
										TailCurlSinStep:=FALSE;
									END_IF	
									TailCurlStep3:=1050;
								END_IF
						END_IF
				1050://左、右压刀开合轴至张开位
						IF NOT TailCurlSinStep THEN					
								IF 	arrAxisCtrl[AxiseNo.AxisName.LeftYDLine].Status.Homed AND arrAxisCtrl[AxiseNo.AxisName.LeftYDLine].Status.NoMoving THEN
									IF arrAxisCtrl[AxiseNo.AxisName.LeftYDLine].Cmd.arrbRealPoint[2] THEN
										arrAxisCtrl[AxiseNo.AxisName.LeftYDLine].Cmd.iGoSetPos:=0;
									ELSE
										arrAxisCtrl[AxiseNo.AxisName.LeftYDLine].Cmd.iGoSetPos:=2;//左压刀开合至张开位
									END_IF
								END_IF					
								IF 	arrAxisCtrl[AxiseNo.AxisName.RightYDLine].Status.Homed AND arrAxisCtrl[AxiseNo.AxisName.RightYDLine].Status.NoMoving THEN
									IF arrAxisCtrl[AxiseNo.AxisName.RightYDLine].Cmd.arrbRealPoint[3] THEN
										arrAxisCtrl[AxiseNo.AxisName.RightYDLine].Cmd.iGoSetPos:=0;
									ELSE
										arrAxisCtrl[AxiseNo.AxisName.RightYDLine].Cmd.iGoSetPos:=3;//右压刀开合至张开位
									END_IF
								END_IF				
								IF arrAxisCtrl[AxiseNo.AxisName.LeftYDLine].Cmd.arrbRealPoint[2] AND arrAxisCtrl[AxiseNo.AxisName.RightYDLine].Cmd.arrbRealPoint[3] THEN
									IF Mach_Control.WJ_b.SinStepMode THEN//尾卷单步模式
										TailCurlSinStep:=TRUE;
									ELSE
										TailCurlSinStep:=FALSE;
									END_IF										
									TailCurlStep3:=1060;
								END_IF	
						END_IF
						
				1060:
						IF NOT TailCurlSinStep THEN		
								IF 	arrAxisCtrl[AxiseNo.AxisName.RightYDUpDown].Status.Homed AND arrAxisCtrl[AxiseNo.AxisName.RightYDUpDown].Status.NoMoving THEN
									IF arrAxisCtrl[AxiseNo.AxisName.RightYDUpDown].Cmd.arrbRealPoint[5] THEN
										arrAxisCtrl[AxiseNo.AxisName.RightYDUpDown].Cmd.iGoSetPos:=0;
									ELSE
										arrAxisCtrl[AxiseNo.AxisName.RightYDUpDown].Cmd.iGoSetPos:=5;//右压好升降上升至下料张开位
									END_IF
								END_IF				
								IF  arrAxisCtrl[AxiseNo.AxisName.RightYDUpDown].Cmd.arrbRealPoint[5] THEN
									IF Mach_Control.WJ_b.SinStepMode THEN//尾卷单步模式
										TailCurlSinStep:=TRUE;
									ELSE
										TailCurlSinStep:=FALSE;
									END_IF	
									TailCurlStep3:=1070;
								END_IF

						END_IF
		
				1065:
					
						(*IF NOT TailCurlSinStep THEN	
							arrCyCtrl[arrCyNo.CylinderName.PreDiaph].Cmd.bON:=TRUE;//叠台压隔膜气缸
							IF arrCyCtrl[arrCyNo.CylinderName.PreDiaph].Status.ONState THEN
								IF Mach_Control.WJ_b.SinStepMode THEN//尾卷单步模式
									TailCurlSinStep:=TRUE;
								ELSE
									TailCurlSinStep:=FALSE;
								END_IF									
								TailCurlStep3:=1070;	
							END_IF	
						END_IF	*)			
									
						
				1070://尾卷夹电芯平移至拉膜位、尾卷夹电芯伸缩至初始位、
						IF NOT TailCurlSinStep THEN	
							tailCult_GearInMultiMaster.Enable:=TRUE;//启动尾卷拉膜凸轮耦合
							fbGearInGMvirbEnable:=TRUE;//尾卷拉膜纠偏
							arrAxisCtrl[AxiseNo.AxisName.TailCurlLine].Cmd.fOverride:=30;
							arrAxisCtrl[AxiseNo.AxisName.TailCurlRetracting].Cmd.fOverride:=30;
							IF  tailCult_GearInMultiMaster.InGear THEN
								
							
										IF 	arrAxisCtrl[AxiseNo.AxisName.TailCurlRetracting].Status.Homed AND arrAxisCtrl[AxiseNo.AxisName.TailCurlRetracting].Status.NoMoving THEN
										
											IF arrAxisCtrl[AxiseNo.AxisName.TailCurlRetracting].Cmd.arrbRealPoint[1] THEN
												arrAxisCtrl[AxiseNo.AxisName.TailCurlRetracting].Cmd.iGoSetPos:=0;
											ELSE
												arrAxisCtrl[AxiseNo.AxisName.TailCurlRetracting].Cmd.iGoSetPos:=1;//尾卷夹电芯伸缩移至初始位
											END_IF
										END_IF				
									
										IF 	arrAxisCtrl[AxiseNo.AxisName.TailCurlLine].Status.Homed AND arrAxisCtrl[AxiseNo.AxisName.TailCurlLine].Status.NoMoving AND
                                               arrAxisCtrl[AxiseNo.AxisName.LCurlingneedleLine].Cmd.arrbRealPoint[1]  AND arrAxisCtrl[AxiseNo.AxisName.SCurlingneedleLine].Cmd.arrbRealPoint[1]  THEN
											IF arrAxisCtrl[AxiseNo.AxisName.TailCurlLine].Cmd.arrbRealPoint[9] THEN
												arrAxisCtrl[AxiseNo.AxisName.TailCurlLine].Cmd.iGoSetPos:=0;
											ELSE
												arrAxisCtrl[AxiseNo.AxisName.TailCurlLine].Cmd.iGoSetPos:=9;//尾卷夹电芯平移至对齐度NG切膜位
											END_IF
										END_IF																		
									IF 	arrAxisCtrl[AxiseNo.AxisName.TailCurlRetracting].Cmd.arrbRealPoint[1] AND arrAxisCtrl[AxiseNo.AxisName.TailCurlLine].Cmd.arrbRealPoint[9]  THEN
											tailCult_GearInMultiMaster.Enable:=FALSE;//启动尾卷拉膜凸轮耦合
											IF Mach_Control.WJ_b.SinStepMode THEN//尾卷单步模式
												TailCurlSinStep:=TRUE;
											ELSE
												TailCurlSinStep:=FALSE;
											END_IF
											fbGearInGMvirbEnable	:=FALSE;
											arrAxisCtrl[AxiseNo.AxisName.TailCurlLine].Cmd.fOverride:=100;
											arrAxisCtrl[AxiseNo.AxisName.TailCurlRetracting].Cmd.fOverride:=100;									
											TailCurlStep3:=1075;
											NGcount:=NGcount+1;
								END_IF	
						END_IF
						END_IF
		

					1075:	
							arrAxisCtrl[AxiseNo.AxisName.TailCurlLine].Cmd.fOverride:=100;
							arrAxisCtrl[AxiseNo.AxisName.TailCurlRetracting].Cmd.fOverride:=100;
							IF NOT TailCurlSinStep THEN			
										IF arrAxis[AxiseNo.AxisName.TailCurlWhirling].Status.Homed AND arrAxisCtrl[AxiseNo.AxisName.TailCurlWhirling].Status.NoMoving THEN
													IF arrAxisCtrl[AxiseNo.AxisName.TailCurlWhirling].Cmd.arrbRealPoint[4] THEN
														arrAxisCtrl[AxiseNo.AxisName.TailCurlWhirling].Cmd.iGoSetPos:=0;
														IF Mach_Control.WJ_b.SinStepMode THEN//尾卷单步模式
															TailCurlSinStep:=TRUE;
														ELSE
															TailCurlSinStep:=FALSE;
														END_IF	
														TailCurlStep3:=1080;
													ELSE
														arrAxisCtrl[AxiseNo.AxisName.TailCurlWhirling].Cmd.iGoSetPos:=4;
													END_IF						
									END_IF
								END_IF
						
	
						
					1080://左、右压刀开合至张开位
						IF NOT TailCurlSinStep THEN		
								
								IF 	arrAxisCtrl[AxiseNo.AxisName.LeftYDUpDown].Status.Homed AND arrAxisCtrl[AxiseNo.AxisName.LeftYDUpDown].Status.NoMoving THEN
									IF arrAxisCtrl[AxiseNo.AxisName.LeftYDUpDown].Cmd.arrbRealPoint[2] THEN
										arrAxisCtrl[AxiseNo.AxisName.LeftYDUpDown].Cmd.iGoSetPos:=0;
									ELSE
										arrAxisCtrl[AxiseNo.AxisName.LeftYDUpDown].Cmd.iGoSetPos:=2;//左压刀升降轴上升至下料高度
									END_IF
								END_IF					
								IF 	arrAxisCtrl[AxiseNo.AxisName.RightYDUpDown].Status.Homed AND arrAxisCtrl[AxiseNo.AxisName.RightYDUpDown].Status.NoMoving THEN
									IF arrAxisCtrl[AxiseNo.AxisName.RightYDUpDown].Cmd.arrbRealPoint[2] THEN
										arrAxisCtrl[AxiseNo.AxisName.RightYDUpDown].Cmd.iGoSetPos:=0;
									ELSE
										arrAxisCtrl[AxiseNo.AxisName.RightYDUpDown].Cmd.iGoSetPos:=2;//右压好升降上升至下料高度
									END_IF
								END_IF																	
								IF 	arrAxisCtrl[AxiseNo.AxisName.TailCurlSEPTAUpDown].Status.Homed AND arrAxisCtrl[AxiseNo.AxisName.TailCurlSEPTAUpDown].Status.NoMoving THEN
									IF arrAxisCtrl[AxiseNo.AxisName.TailCurlSEPTAUpDown].Cmd.arrbRealPoint[2] THEN
										arrAxisCtrl[AxiseNo.AxisName.TailCurlSEPTAUpDown].Cmd.iGoSetPos:=0;
									ELSE
										arrAxisCtrl[AxiseNo.AxisName.TailCurlSEPTAUpDown].Cmd.iGoSetPos:=2;//
									END_IF
								END_IF					
								IF 	arrAxisCtrl[AxiseNo.AxisName.TailCurlUpDown].Status.Homed AND arrAxisCtrl[AxiseNo.AxisName.TailCurlUpDown].Status.NoMoving THEN
									IF arrAxisCtrl[AxiseNo.AxisName.TailCurlUpDown].Cmd.arrbRealPoint[2] THEN
										arrAxisCtrl[AxiseNo.AxisName.TailCurlUpDown].Cmd.iGoSetPos:=0;
									ELSE
										arrAxisCtrl[AxiseNo.AxisName.TailCurlUpDown].Cmd.iGoSetPos:=2;//
									END_IF
								END_IF									
								
								IF  arrAxisCtrl[AxiseNo.AxisName.TailCurlUpDown].Cmd.arrbRealPoint[2] AND arrAxisCtrl[AxiseNo.AxisName.TailCurlSEPTAUpDown].Cmd.arrbRealPoint[2] AND
									arrAxisCtrl[AxiseNo.AxisName.LeftYDUpDown].Cmd.arrbRealPoint[2] AND arrAxisCtrl[AxiseNo.AxisName.RightYDUpDown].Cmd.arrbRealPoint[2]  THEN
									IF Mach_Control.WJ_b.SinStepMode THEN//尾卷单步模式
										TailCurlSinStep:=TRUE;
									ELSE
										TailCurlSinStep:=FALSE;
									END_IF		
									TailCurlStep3:=1085;
								END_IF
						END_IF		
				1085:
						IF NOT TailCurlSinStep THEN	
							arrCyCtrl[arrCyNo.ElectValveName.PoleSplintVacuum_D].Cmd.bON:=TRUE;//夹膜下夹板真空	
							arrCyCtrl[arrCyNo.CylinderName.PoleSplintCy_D].Cmd.bON:=TRUE;//夹膜下夹板上升
								IF arrCyCtrl[arrCyNo.CylinderName.PoleSplintCy_D].Status.ONState THEN
									IF Mach_Control.WJ_b.SinStepMode THEN//尾卷单步模式
										TailCurlSinStep:=TRUE;
									ELSE
										TailCurlSinStep:=FALSE;
									END_IF									
									TailCurlStep3:=1090;	
								END_IF	
						END_IF	
	
				1090:
					
						IF NOT TailCurlSinStep THEN	
							arrCyCtrl[arrCyNo.CylinderName.PreDiaph].Cmd.bON:=TRUE;//叠台压隔膜气缸
							IF arrCyCtrl[arrCyNo.CylinderName.PreDiaph].Status.ONState THEN
								IF Mach_Control.WJ_b.SinStepMode THEN//尾卷单步模式
									TailCurlSinStep:=TRUE;
								ELSE
									TailCurlSinStep:=FALSE;
								END_IF									
								TailCurlStep3:=1100;
							END_IF	
						END_IF							
			


				1100://左、右压刀开合移至初始位，叠台上升至初始位
						IF NOT TailCurlSinStep THEN		
									IF 	arrAxisCtrl[AxiseNo.AxisName.LeftYDLine].Status.Homed AND arrAxisCtrl[AxiseNo.AxisName.LeftYDLine].Status.NoMoving THEN
										IF arrAxisCtrl[AxiseNo.AxisName.LeftYDLine].Cmd.arrbRealPoint[1] THEN
											arrAxisCtrl[AxiseNo.AxisName.LeftYDLine].Cmd.iGoSetPos:=0;
										ELSE
											arrAxisCtrl[AxiseNo.AxisName.LeftYDLine].Cmd.iGoSetPos:=1;//左压刀开合至初始位
										END_IF
									END_IF					
									IF 	arrAxisCtrl[AxiseNo.AxisName.RightYDLine].Status.Homed AND arrAxisCtrl[AxiseNo.AxisName.RightYDLine].Status.NoMoving THEN
										IF arrAxisCtrl[AxiseNo.AxisName.RightYDLine].Cmd.arrbRealPoint[1] THEN
											arrAxisCtrl[AxiseNo.AxisName.RightYDLine].Cmd.iGoSetPos:=0;
										ELSE
											arrAxisCtrl[AxiseNo.AxisName.RightYDLine].Cmd.iGoSetPos:=1;//右压刀开合至初始位
										END_IF
									END_IF
									IF 	arrAxisCtrl[AxiseNo.AxisName.DTUpDown].Status.Homed AND arrAxisCtrl[AxiseNo.AxisName.DTUpDown].Status.NoMoving THEN
										IF arrAxisCtrl[AxiseNo.AxisName.DTUpDown].Cmd.arrbRealPoint[1] THEN
											arrAxisCtrl[AxiseNo.AxisName.DTUpDown].Cmd.iGoSetPos:=0;
										ELSE
											arrAxisCtrl[AxiseNo.AxisName.DTUpDown].Cmd.iGoSetPos:=1;//叠台升降上升至初始位
										END_IF
									END_IF
									IF 	arrAxisCtrl[AxiseNo.AxisName.LeftYDLine].Cmd.arrbRealPoint[1] AND arrAxisCtrl[AxiseNo.AxisName.RightYDLine].Cmd.arrbRealPoint[1] AND 
										arrAxisCtrl[AxiseNo.AxisName.DTUpDown].Cmd.arrbRealPoint[1] THEN
												TailCurlStep3:=1110;
												IF Mach_Control.WJ_b.SinStepMode THEN//尾卷单步模式
													TailCurlSinStep:=TRUE;
												ELSE
													TailCurlSinStep:=FALSE;
												END_IF	
									END_IF	
						END_IF
				
					



				1110://左、右压刀升降下降至初始位，压隔膜
						IF NOT TailCurlSinStep THEN			
									IF 	arrAxisCtrl[AxiseNo.AxisName.LeftYDUpDown].Status.Homed AND arrAxisCtrl[AxiseNo.AxisName.LeftYDUpDown].Status.NoMoving THEN
										IF arrAxisCtrl[AxiseNo.AxisName.LeftYDUpDown].Cmd.arrbRealPoint[1] THEN
											arrAxisCtrl[AxiseNo.AxisName.LeftYDUpDown].Cmd.iGoSetPos:=0;
										ELSE
											arrAxisCtrl[AxiseNo.AxisName.LeftYDUpDown].Cmd.iGoSetPos:=1;//左压刀升降轴下降至初始高度
										END_IF
									END_IF					
									IF 	arrAxisCtrl[AxiseNo.AxisName.RightYDUpDown].Status.Homed AND arrAxisCtrl[AxiseNo.AxisName.RightYDUpDown].Status.NoMoving THEN
										IF arrAxisCtrl[AxiseNo.AxisName.RightYDUpDown].Cmd.arrbRealPoint[1] THEN
											arrAxisCtrl[AxiseNo.AxisName.RightYDUpDown].Cmd.iGoSetPos:=0;
										ELSE
											arrAxisCtrl[AxiseNo.AxisName.RightYDUpDown].Cmd.iGoSetPos:=1;//右压好升降下降至初始高度
										END_IF
									END_IF				
									IF arrAxisCtrl[AxiseNo.AxisName.LeftYDUpDown].Cmd.arrbRealPoint[1] AND arrAxisCtrl[AxiseNo.AxisName.RightYDUpDown].Cmd.arrbRealPoint[1] THEN
										IF Mach_Control.WJ_b.SinStepMode THEN//尾卷单步模式
											TailCurlSinStep:=TRUE;
										ELSE
											TailCurlSinStep:=FALSE;
										END_IF											
										TailCurlStep3:=1120;
										hot_time_ton.IN:=FALSE;
									END_IF
						END_IF
						
					(*1120:
						Mach_Control.WJ_b.HotCut:=TRUE;//启动热切
						WJ_TON[1].IN:=TRUE;
						TailCurlStep3:=1130;		
					
						
				1130://热切丝加热、热切升降气缸下降，切隔膜///////////////////////////////
					IF NOT TailCurlSinStep THEN	
					arrCyCtrl[arrCyNo.CylinderName.PoleHotCutterCy].Cmd.bON:=TRUE;//隔膜热切升降气缸伸出
								IF arrCyCtrl[arrCyNo.CylinderName.PoleHotCutterCy].Status.ONState  THEN
										Mach_Control.WJ_b.HotCut:=FALSE;//启动热切
						                WJ_TON[1].IN:=FALSE;
							IF Mach_Control.WJ_b.SinStepMode THEN//尾卷单步模式
								TailCurlSinStep:=TRUE;
							ELSE
								TailCurlSinStep:=FALSE;
							END_IF							
									TailCurlStep3:=1140;	
								END_IF	
					END_IF*)	
				
				1140://热切升降气缸下降/////////////////////////////////////////
				IF NOT TailCurlSinStep THEN	
					Blueflaging:=FALSE;
					arrCyCtrl[arrCyNo.CylinderName.PoleHotCutterCy].Cmd.bOFF:=TRUE;//隔膜热切升降气缸缩回	
						IF arrCyCtrl[arrCyNo.CylinderName.PoleHotCutterCy].Status.OFFState THEN
							IF Mach_Control.WJ_b.SinStepMode THEN//尾卷单步模式
								TailCurlSinStep:=TRUE;
							ELSE
								TailCurlSinStep:=FALSE;
							END_IF									
							TailCurlStep3:=1142;	
						END_IF	
				END_IF	

				1142://叠台真空打开
					arrCyCtrl[arrCyNo.ElectValveName.DTVacuum].Cmd.bON:=TRUE;
					arrCyCtrl[arrCyNo.ElectValveName.DTVacuum].Cmd.bOFF:=FALSE;
					TailCurlStep3:=1145;
					
				1145:
						IF NOT TailCurlSinStep THEN	
							arrCyCtrl[arrCyNo.ElectValveName.PoleSplintVacuum_D].Cmd.bOFF:=TRUE;//夹膜下夹板真空	
							arrCyCtrl[arrCyNo.CylinderName.PoleSplintCy_D].Cmd.bOFF:=TRUE;//夹膜下夹板上升
								IF arrCyCtrl[arrCyNo.CylinderName.PoleSplintCy_D].Status.OFFState THEN
									IF Mach_Control.WJ_b.SinStepMode THEN//尾卷单步模式
										TailCurlSinStep:=TRUE;
									ELSE
										TailCurlSinStep:=FALSE;
									END_IF									
									TailCurlStep3:=1148;	
								END_IF	
						END_IF							
				
				1148:
					IF 	arrAxisCtrl[AxiseNo.AxisName.TailCurlSEPTAUpDown].Status.Homed AND arrAxisCtrl[AxiseNo.AxisName.TailCurlSEPTAUpDown].Status.NoMoving THEN
						IF arrAxisCtrl[AxiseNo.AxisName.TailCurlSEPTAUpDown].Cmd.arrbRealPoint[1] THEN
							arrAxisCtrl[AxiseNo.AxisName.TailCurlSEPTAUpDown].Cmd.iGoSetPos:=0;
						ELSE
							arrAxisCtrl[AxiseNo.AxisName.TailCurlSEPTAUpDown].Cmd.iGoSetPos:=1;//
						END_IF
					END_IF
					IF arrAxisCtrl[AxiseNo.AxisName.TailCurlSEPTAUpDown].Cmd.arrbRealPoint[1] THEN
						TailCurlStep3:=1150;	
					END_IF
	

				1150:
					CellMemory[Mach_Control.WJ_b.WJ_Memory]:=CellMemory[Mach_Control.DT_b.DT_Memory];
					MEMSET(ADR(CellMemory[Mach_Control.DT_b.DT_Memory]),0,SIZEOF(CellMemory[Mach_Control.DT_b.DT_Memory]));
					TailCurlStep3:=1160;
		
				1160:
					
						IF NOT TailCurlSinStep THEN	
							arrCyCtrl[arrCyNo.CylinderName.PreDiaph].Cmd.bOFF:=TRUE;//
							IF arrCyCtrl[arrCyNo.CylinderName.PreDiaph].Status.OFFState THEN
								IF Mach_Control.WJ_b.SinStepMode THEN//尾卷单步模式
									TailCurlSinStep:=TRUE;
								ELSE
									TailCurlSinStep:=FALSE;
								END_IF									
								TailCurlStep3:=1170;
								TailCurlStep6:=10;//启动判断夹膜平移是否已经在安全位置叠台下料完成	
							END_IF	
						END_IF

				1170:
					IF NOT TailCurlSinStep THEN	
					
						IF 	arrAxisCtrl[AxiseNo.AxisName.TailCurlLine].Status.Homed AND arrAxisCtrl[AxiseNo.AxisName.TailCurlLine].Status.NoMoving AND
                                arrAxisCtrl[AxiseNo.AxisName.LCurlingneedleLine].Cmd.arrbRealPoint[1]  AND arrAxisCtrl[AxiseNo.AxisName.SCurlingneedleLine].Cmd.arrbRealPoint[1] AND
                                 arrAxisCtrl[AxiseNo.AxisName.TailCurlWhirling].Cmd.arrbRealPoint[1]  THEN
								IF arrAxisCtrl[AxiseNo.AxisName.TailCurlLine].Cmd.arrbRealPoint[1] THEN
									arrAxisCtrl[AxiseNo.AxisName.TailCurlLine].Cmd.iGoSetPos:=0;
								ELSE
									arrAxisCtrl[AxiseNo.AxisName.TailCurlLine].Cmd.iGoSetPos:=1;//尾卷夹电芯平移至初始位
								END_IF
							END_IF	
						IF   arrAxis[AxiseNo.AxisName.TailCurlSEPTALine].Status.Homed AND arrAxisCtrl[AxiseNo.AxisName.TailCurlSEPTALine].Status.NoMoving AND arrAxisCtrl[AxiseNo.AxisName.TailCurlLine].Status.Homed 
								AND arrAxisCtrl[AxiseNo.AxisName.TailCurlLine].Status.fActPos<arrAxisPar[AxiseNo.AxisName.TailCurlLine].arrTargetPoint[7] THEN
								IF arrAxisCtrl[AxiseNo.AxisName.TailCurlSEPTALine].Cmd.arrbRealPoint[1] THEN
									arrAxisCtrl[AxiseNo.AxisName.TailCurlSEPTALine].Cmd.iGoSetPos:=0;
								ELSE
									arrAxisCtrl[AxiseNo.AxisName.TailCurlSEPTALine].Cmd.iGoSetPos:=1;//尾卷夹隔膜平移至初始位
								END_IF
						END_IF
						IF arrAxisCtrl[AxiseNo.AxisName.TailCurlLine].Cmd.arrbRealPoint[1] AND arrAxisCtrl[AxiseNo.AxisName.TailCurlLine].Status.NoMoving 
							AND arrAxisCtrl[AxiseNo.AxisName.TailCurlSEPTALine].Cmd.arrbRealPoint[1] AND  arrAxisCtrl[AxiseNo.AxisName.TailCurlSEPTALine].Status.NoMoving AND
							TailCurlStep6=666  THEN
								IF Mach_Control.WJ_b.SinStepMode THEN//尾卷单步模式
									TailCurlSinStep:=TRUE;
								ELSE
									TailCurlSinStep:=FALSE;
								END_IF									
								TailCurlStep3:=1180;
							END_IF
					END_IF
				1180://尾卷夹电芯升降至下电芯位      
						  IF NOT TailCurlSinStep THEN		                                                                                                                                                                                                                                                                                                                                                                                                   		
									IF arrAxisCtrl[AxiseNo.AxisName.TailCurlUpDown].Status.Homed AND arrAxisCtrl[AxiseNo.AxisName.TailCurlUpDown].Status.NoMoving THEN
										IF arrAxisCtrl[AxiseNo.AxisName.TailCurlUpDown].Cmd.arrbRealPoint[3] THEN
											arrAxisCtrl[AxiseNo.AxisName.TailCurlUpDown].Cmd.iGoSetPos:=0;	
										ELSE
											arrAxisCtrl[AxiseNo.AxisName.TailCurlUpDown].Cmd.iGoSetPos:=3;//尾卷夹电芯升降至下电芯位
										END_IF
									END_IF
							IF 	arrAxisCtrl[AxiseNo.AxisName.TailCurlSEPTAUpDown].Status.Homed AND arrAxisCtrl[AxiseNo.AxisName.TailCurlSEPTAUpDown].Status.NoMoving THEN
								IF arrAxisCtrl[AxiseNo.AxisName.TailCurlSEPTAUpDown].Cmd.arrbRealPoint[1] THEN
									arrAxisCtrl[AxiseNo.AxisName.TailCurlSEPTAUpDown].Cmd.iGoSetPos:=0;
								ELSE
									arrAxisCtrl[AxiseNo.AxisName.TailCurlSEPTAUpDown].Cmd.iGoSetPos:=1;
								END_IF
							END_IF
							IF arrAxisCtrl[AxiseNo.AxisName.TailCurlUpDown].Cmd.arrbRealPoint[3] AND arrAxisCtrl[AxiseNo.AxisName.TailCurlUpDown].Status.NoMoving
								AND arrAxisCtrl[AxiseNo.AxisName.TailCurlSEPTAUpDown].Cmd.arrbRealPoint[1] AND  arrAxisCtrl[AxiseNo.AxisName.TailCurlSEPTAUpDown].Status.NoMoving THEN
								IF Mach_Control.WJ_b.SinStepMode THEN//尾卷单步模式
												TailCurlSinStep:=TRUE;
											ELSE
												TailCurlSinStep:=FALSE;
											END_IF									
											TailCurlStep3:=1190;
							END_IF	
						END_IF
						
						
						
				1190://尾卷夹电芯旋转至下电芯位
						IF NOT TailCurlSinStep THEN				
								IF 	(*arrCyCtrl[arrCyNo.CylinderName.TailCurlSplintCy].Status.ONState AND*)  arrAxisCtrl[AxiseNo.AxisName.TailCurlLine].Status.Homed 
									AND arrAxisCtrl[AxiseNo.AxisName.TailCurlLine].Status.NoMoving AND arrAxisCtrl[AxiseNo.AxisName.GluingLine].Status.Homed AND
									arrAxisCtrl[AxiseNo.AxisName.GluingLine].Status.fActPos<=arrAxispar[AxiseNo.AxisName.GluingLine].arrTargetPoint[10] 
									AND NOT Mach_Control.TJ_b.StickerFlag  THEN
									IF arrAxisCtrl[AxiseNo.AxisName.TailCurlWhirling].Cmd.arrbRealPoint[2] THEN
										arrAxisCtrl[AxiseNo.AxisName.TailCurlWhirling].Cmd.iGoSetPos:=0;
											IF Mach_Control.WJ_b.SinStepMode THEN//尾卷单步模式
												TailCurlSinStep:=TRUE;
											ELSE
												TailCurlSinStep:=FALSE;
											END_IF										
										TailCurlStep3:=1200;
									ELSE
										arrAxisCtrl[AxiseNo.AxisName.TailCurlWhirling].Cmd.iGoSetPos:=2;//尾卷夹电芯平移至下电芯位
									END_IF
								END_IF
						END_IF		
						
				
						
			
				1200:
				//尾卷夹电芯去下料避让位   
						  IF NOT TailCurlSinStep THEN		                                                                                                                                                                                                                                                                                                                                                                                                   		
									IF arrAxisCtrl[AxiseNo.AxisName.TailCurlLine].Status.Homed AND arrAxisCtrl[AxiseNo.AxisName.TailCurlLine].Status.NoMoving THEN
										IF arrAxisCtrl[AxiseNo.AxisName.TailCurlLine].Cmd.arrbRealPoint[10] THEN
											arrAxisCtrl[AxiseNo.AxisName.TailCurlLine].Cmd.iGoSetPos:=0;
											IF Mach_Control.WJ_b.SinStepMode THEN//尾卷单步模式
												TailCurlSinStep:=TRUE;
											ELSE
												TailCurlSinStep:=FALSE;
											END_IF									
											TailCurlStep3:=1210;
										ELSE
											arrAxisCtrl[AxiseNo.AxisName.TailCurlLine].Cmd.iGoSetPos:=10;//尾卷夹电芯平移至避让位
										END_IF
									END_IF
							END_IF
				1210:
						IF NOT TailCurlSinStep THEN
								Mach_Control.WJ_b.TailCultOffloading:=TRUE;//下电芯请求														
								TailCurlStep3:=1220;
								
								IF Mach_Control.WJ_b.SinStepMode THEN//尾卷单步模式
									TailCurlSinStep:=TRUE;
								ELSE
									TailCurlSinStep:=FALSE;
								END_IF					
						END_IF				
						

				1220:   ///////////////////
						
					IF 	arrAxisCtrl[AxiseNo.AxisName.GluingLine].Cmd.arrbRealPoint[8] AND arrAxisCtrl[AxiseNo.AxisName.GluingLine].Status.NoMoving
						AND arrAxisCtrl[AxiseNo.AxisName.GluingWhirling].Cmd.arrbRealPoint[5] AND arrAxisCtrl[AxiseNo.AxisName.GluingWhirling].Status.NoMoving
						AND arrCyCtrl[arrCyNo.CylinderName.PullGlueModelCy].Status.ONState AND NOT arrCyCtrl[arrCyNo.CylinderName.PullGlueModelCy].Status.Error2 
						AND arrAxisCtrl[AxiseNo.AxisName.TailCurlLine].Status.Homed AND arrAxisCtrl[AxiseNo.AxisName.TailCurlLine].Status.NoMoving	
						AND NOT Mach_Control.TJ_b.StickerDone  AND NOT Mach_Control.TJ_b.StickerFlag
						AND NOT CellMemory[Mach_Control.TJ_b.TJ_Memory].Cell AND NOT Mach_Control.se.GluebHave	THEN
						TailCurlStep3:=1225;
					ELSIF Mach_Control.se.GluebHave AND arrAxisCtrl[AxiseNo.AxisName.GluingWhirling].Status.NoMoving THEN
						Mach_Control.TJ_b.Error[9]:=TRUE; //贴胶夹爪有信号无记忆报警
					END_IF
						
				1225:
						IF arrAxisCtrl[AxiseNo.AxisName.TailCurlLine].Cmd.arrbRealPoint[6] THEN
							arrAxisCtrl[AxiseNo.AxisName.TailCurlLine].Cmd.iGoSetPos:=0;
							IF Mach_Control.WJ_b.SinStepMode THEN//尾卷单步模式
								TailCurlSinStep:=TRUE;
							ELSE
								TailCurlSinStep:=FALSE;
							END_IF									
							TailCurlStep3:=1230;
						ELSE
							arrAxisCtrl[AxiseNo.AxisName.TailCurlLine].Cmd.iGoSetPos:=6;//尾卷夹电芯平移至下电芯位
						END_IF
						
						
				1230:
							IF NOT TailCurlSinStep THEN		
									IF 	arrAxisCtrl[AxiseNo.AxisName.GluingLine].Cmd.arrbRealPoint[8] AND arrAxisCtrl[AxiseNo.AxisName.GluingLine].Status.NoMoving
										AND arrAxisCtrl[AxiseNo.AxisName.GluingWhirling].Cmd.arrbRealPoint[5] AND arrAxisCtrl[AxiseNo.AxisName.GluingWhirling].Status.NoMoving
										AND arrCyCtrl[arrCyNo.CylinderName.PullGlueModelCy].Status.ONState AND NOT arrCyCtrl[arrCyNo.CylinderName.PullGlueModelCy].Status.Error2 
										AND arrAxisCtrl[AxiseNo.AxisName.TailCurlRetracting].Status.Homed AND arrAxisCtrl[AxiseNo.AxisName.TailCurlRetracting].Status.NoMoving		THEN
									IF arrAxisCtrl[AxiseNo.AxisName.TailCurlRetracting].Cmd.arrbRealPoint[3] THEN
										arrAxisCtrl[AxiseNo.AxisName.TailCurlRetracting].Cmd.iGoSetPos:=0;
										IF Mach_Control.WJ_b.SinStepMode THEN//尾卷单步模式
											TailCurlSinStep:=TRUE;
										ELSE
											TailCurlSinStep:=FALSE;
										END_IF									
										TailCurlStep3:=1240;
									ELSE
										arrAxisCtrl[AxiseNo.AxisName.TailCurlRetracting].Cmd.iGoSetPos:=3;//尾卷夹电芯伸缩至下电芯位
										END_IF
									END_IF
							END_IF	
				1240:
							IF NOT TailCurlSinStep THEN			
								IF 	arrAxisCtrl[AxiseNo.AxisName.TailCurlUpDown].Status.Homed AND arrAxisCtrl[AxiseNo.AxisName.TailCurlUpDown].Status.NoMoving  THEN
									IF arrAxisCtrl[AxiseNo.AxisName.TailCurlUpDown].Cmd.arrbRealPoint[4] THEN
													arrAxisCtrl[AxiseNo.AxisName.TailCurlUpDown].Cmd.iGoSetPos:=0;
													IF Mach_Control.WJ_b.SinStepMode THEN//尾卷单步模式
													TailCurlSinStep:=TRUE;
													ELSE
														TailCurlSinStep:=FALSE;
													END_IF	
													TailCurlStep3:=1260;
									ELSE
													arrAxisCtrl[AxiseNo.AxisName.TailCurlUpDown].Cmd.iGoSetPos:=4;//尾卷夹电芯升降至下电芯位
									END_IF
								END_IF	
						END_IF									
(*						
				1250:
				
						IF NOT TailCurlSinStep THEN				
							arrCyCtrl[arrCyNo.CylinderName.PullGlueModelCy].Cmd.bOFF:=TRUE;//贴胶治具气缸闭合
							IF arrCyCtrl[arrCyNo.CylinderName.PullGlueModelCy].Status.OFFState THEN
								IF Mach_Control.WJ_b.SinStepMode THEN//尾卷单步模式
									TailCurlSinStep:=TRUE;
								ELSE
									TailCurlSinStep:=FALSE;
								END_IF										
								TailCurlStep3:=1260;
							END_IF
						END_IF
*)

				1260:
				

					IF NOT TailCurlSinStep THEN				
							arrCyCtrl[arrCyNo.CylinderName.TailCurlSplintCy].Cmd.bOFF:=TRUE;//尾卷夹爪气缸打开
							IF arrCyCtrl[arrCyNo.CylinderName.TailCurlSplintCy].Status.OFFState THEN
								IF Mach_Control.WJ_b.SinStepMode THEN//尾卷单步模式
									TailCurlSinStep:=TRUE;
								ELSE
									TailCurlSinStep:=FALSE;
								END_IF	
								Mach_Control.TJ_b.StickerFlag:=TRUE;//置位贴胶夹爪有料标记
								TailCurlStep3:=1265;
							END_IF
						END_IF

				1265:
					IF NOT TailCurlSinStep THEN			
						IF 	arrAxisCtrl[AxiseNo.AxisName.TailCurlUpDown].Status.Homed AND arrAxisCtrl[AxiseNo.AxisName.TailCurlUpDown].Status.NoMoving  AND
							arrAxisCtrl[AxiseNo.AxisName.TailCurlUpDown].Cmd.arrbRealPoint[4] THEN
							arrAxisPar[AxiseNo.AxisName.TailCurlUpDown].fVelocity_of_Rel := 20   ;
							arrAxisCtrl[AxiseNo.AxisName.TailCurlUpDown].Cmd.fPosition_of_Rel :=3 ;
							arrAxisCtrl[AxiseNo.AxisName.TailCurlUpDown].Cmd.bMoveRel :=  TRUE ;
						END_IF
							IF arrAxis[AxiseNo.AxisName.TailCurlUpDown].NcToPlc.SetPos-arrAxisPar[AxiseNo.AxisName.TailCurlUpDown].arrTargetPoint[4] >=3  
							AND arrAxisCtrl[AxiseNo.AxisName.TailCurlUpDown].Status.NoMoving THEN
								IF Mach_Control.WJ_b.SinStepMode THEN//尾卷单步模式
									TailCurlSinStep:=TRUE;
								ELSE
									TailCurlSinStep:=FALSE;
								END_IF
								TailCurlStep3:=1270;
							END_IF
					END_IF	
									
							
				1270:// 尾卷夹电芯平移至下料避让位
						IF NOT TailCurlSinStep THEN			
								IF 	arrAxisCtrl[AxiseNo.AxisName.TailCurlLine].Status.Homed AND arrAxisCtrl[AxiseNo.AxisName.TailCurlLine].Status.NoMoving THEN
									IF arrAxisCtrl[AxiseNo.AxisName.TailCurlLine].Cmd.arrbRealPoint[10] THEN
										arrAxisCtrl[AxiseNo.AxisName.TailCurlLine].Cmd.iGoSetPos:=0;
									IF Mach_Control.WJ_b.SinStepMode THEN//尾卷单步模式
									TailCurlSinStep:=TRUE;
								ELSE
									TailCurlSinStep:=FALSE;
								END_IF	
										TailCurlStep3:=1280;
									ELSE
										arrAxisCtrl[AxiseNo.AxisName.TailCurlLine].Cmd.iGoSetPos:=10;//尾卷夹电芯平移至下料避让位
									END_IF
								END_IF	
						END_IF	



				1280:	
					CellMemory[Mach_Control.TJ_b.TJ_Memory]:=CellMemory[Mach_Control.WJ_b.WJ_Memory];
					MEMSET(ADR(CellMemory[Mach_Control.WJ_b.WJ_Memory]),0,SIZEOF(CellMemory[Mach_Control.WJ_b.WJ_Memory]));		
					TailCurlStep3:=1290;		
						
						
						
						
						
						
						
				1290:
		
						IF NOT TailCurlSinStep THEN			
								IF 	arrAxisCtrl[AxiseNo.AxisName.TailCurlRetracting].Status.Homed AND arrAxisCtrl[AxiseNo.AxisName.TailCurlRetracting].Status.NoMoving THEN
									IF arrAxisCtrl[AxiseNo.AxisName.TailCurlRetracting].Cmd.arrbRealPoint[1] THEN
										arrAxisCtrl[AxiseNo.AxisName.TailCurlRetracting].Cmd.iGoSetPos:=0;
										IF Mach_Control.WJ_b.SinStepMode THEN//尾卷单步模式
									TailCurlSinStep:=TRUE;
								ELSE
									TailCurlSinStep:=FALSE;
								END_IF	
										
										TailCurlStep3:=1300;
									ELSE
										arrAxisCtrl[AxiseNo.AxisName.TailCurlRetracting].Cmd.iGoSetPos:=1;//尾卷夹电芯伸缩回到初始位
									END_IF
								END_IF	
						END_IF	
						
						
						
						
				1300:
				IF NOT TailCurlSinStep THEN		
					 IF arrAxisCtrl[AxiseNo.AxisName.GluingLine].Status.fActPos<=arrAxispar[AxiseNo.AxisName.GluingLine].arrTargetPoint[10] 
						AND arrAxisCtrl[AxiseNo.AxisName.GluingLine].Status.Homed AND NOT Mach_Control.WJ_b.TailCultOffloading AND arrAxisCtrl[AxiseNo.AxisName.TailCurlLine].Status.Homed 
						AND arrAxisCtrl[AxiseNo.AxisName.TailCurlLine].Status.NoMoving THEN
						
								IF arrAxisCtrl[AxiseNo.AxisName.TailCurlLine].Cmd.arrbRealPoint[1] THEN
									IF Mach_Control.WJ_b.SinStepMode THEN//尾卷单步模式
									TailCurlSinStep:=TRUE;
								ELSE
									TailCurlSinStep:=FALSE;
								END_IF	
									arrAxisCtrl[AxiseNo.AxisName.TailCurlLine].Cmd.iGoSetPos:=0;
									//Mach_Control.WJ_b.TailCultOffloadingDone:=TRUE;
									TailCurlStep3:=1305;
								ELSE
									arrAxisCtrl[AxiseNo.AxisName.TailCurlLine].Cmd.iGoSetPos:=1;//尾卷夹电芯平移至初始位
								END_IF
						END_IF	
				END_IF	

				1305:
							IF NOT TailCurlSinStep THEN			
								IF 	arrAxisCtrl[AxiseNo.AxisName.TailCurlUpDown].Status.Homed AND arrAxisCtrl[AxiseNo.AxisName.TailCurlUpDown].Status.NoMoving  THEN
									IF arrAxisCtrl[AxiseNo.AxisName.TailCurlUpDown].Cmd.arrbRealPoint[4] THEN
													arrAxisCtrl[AxiseNo.AxisName.TailCurlUpDown].Cmd.iGoSetPos:=0;
													IF Mach_Control.WJ_b.SinStepMode THEN//尾卷单步模式
													TailCurlSinStep:=TRUE;
													ELSE
														TailCurlSinStep:=FALSE;
													END_IF	
													TailCurlStep3:=1310;
									ELSE
													arrAxisCtrl[AxiseNo.AxisName.TailCurlUpDown].Cmd.iGoSetPos:=4;//尾卷夹电芯升降至下电芯位
									END_IF
								END_IF	
						END_IF	
				
				1310:
					IF NOT TailCurlSinStep THEN		
					 IF arrAxisCtrl[AxiseNo.AxisName.GluingLine].Status.fActPos<=arrAxispar[AxiseNo.AxisName.GluingLine].arrTargetPoint[10] 
						AND arrAxisCtrl[AxiseNo.AxisName.GluingLine].Status.Homed AND NOT Mach_Control.WJ_b.TailCultOffloading AND arrAxis[AxiseNo.AxisName.TailCurlWhirling].Status.Homed 
						AND arrAxisCtrl[AxiseNo.AxisName.TailCurlWhirling].Status.NoMoving AND arrAxisCtrl[AxiseNo.AxisName.TailCurlLine].Status.NoMoving AND arrAxisCtrl[AxiseNo.AxisName.TailCurlLine].Cmd.arrbRealPoint[1] THEN
						
								IF arrAxisCtrl[AxiseNo.AxisName.TailCurlWhirling].Cmd.arrbRealPoint[1] THEN
									IF Mach_Control.WJ_b.SinStepMode THEN//尾卷单步模式
									TailCurlSinStep:=TRUE;
								ELSE
									TailCurlSinStep:=FALSE;
								END_IF	
									arrAxisCtrl[AxiseNo.AxisName.TailCurlWhirling].Cmd.iGoSetPos:=0;
									
									TailCurlStep3:=1320;
								ELSE
									arrAxisCtrl[AxiseNo.AxisName.TailCurlWhirling].Cmd.iGoSetPos:=1;//尾卷夹电芯旋转至取电芯位
								END_IF
						END_IF	
				END_IF	
	
	            1320://尾卷夹电芯平移去取电芯等待位
					 IF NOT TailCurlSinStep THEN	
								 IF  arrAxisCtrl[AxiseNo.AxisName.TailCurlUpDown].Status.Homed AND arrAxisCtrl[AxiseNo.AxisName.TailCurlUpDown].Status.NoMoving THEN
												IF arrAxisCtrl[AxiseNo.AxisName.TailCurlUpDown].Cmd.arrbRealPoint[1] THEN
													arrAxisCtrl[AxiseNo.AxisName.TailCurlUpDown].Cmd.iGoSetPos:=0;
												ELSE
													arrAxisCtrl[AxiseNo.AxisName.TailCurlUpDown].Cmd.iGoSetPos:=1;//尾卷夹升降去取电芯高度
												END_IF
								 END_IF
							 
							   IF arrAxisCtrl[AxiseNo.AxisName.TailCurlWhirling].Cmd.arrbRealPoint[1] AND arrAxisCtrl[AxiseNo.AxisName.TailCurlUpDown].Cmd.arrbRealPoint[1] AND
								  arrAxisCtrl[AxiseNo.AxisName.TailCurlSEPTALine].Cmd.arrbRealPoint[1] AND  arrAxisCtrl[AxiseNo.AxisName.TailCurlSEPTAUpDown].Cmd.arrbRealPoint[1] AND
								  arrAxisCtrl[AxiseNo.AxisName.LCurlingneedleLine].Cmd.arrbRealPoint[1] AND arrAxisCtrl[AxiseNo.AxisName.SCurlingneedleLine].Cmd.arrbRealPoint[1] AND
								  arrCyCtrl[arrCyNo.CylinderName.PoleSplintCy_D].Io.DIOFFSwitch AND arrCyCtrl[arrCyNo.CylinderName.TailCurlUpdownCy].Io.DIOFFSwitch AND
								  arrAxisCtrl[AxiseNo.AxisName.TailCurlLine].Status.Homed AND arrAxisCtrl[AxiseNo.AxisName.TailCurlLine].Status.NoMoving  THEN
									   IF arrAxisCtrl[AxiseNo.AxisName.TailCurlLine].Cmd.arrbRealPoint[11]  THEN
										  arrAxisCtrl[AxiseNo.AxisName.TailCurlLine].Cmd.iGoSetPos:=0;
											IF Mach_Control.WJ_b.SinStepMode THEN//尾卷单步模式
											   TailCurlSinStep:=TRUE;
											ELSE
											   TailCurlSinStep:=FALSE;
											END_IF									
											   TailCurlStep3:=0;
											   TailCurlTorMark:=FALSE;//尾卷夹电芯平移力矩判断标志位
									   ELSE
										   arrAxisCtrl[AxiseNo.AxisName.TailCurlLine].Cmd.iGoSetPos:=11;//尾卷夹电芯平移去取电芯等待位
										   TailCurlTorMark:=TRUE;//尾卷夹电芯平移力矩判断标志位
									   END_IF   
								END_IF
					  END_IF
	
	
	END_CASE	
ELSE
	//tailCult_GearInMultiMaster.Enable:=FALSE;//尾卷拉膜耦合放卷虚轴
//	tailCurlGearInEnable:=FALSE;//夹电芯平移轴与夹隔膜平移轴电子齿轮耦合
//	fbGearInGMvirbEnable	:=FALSE;	//隔膜纠䐔
;
END_IF	

CASE TailCurlStep3 OF 
	
		

	   200:
	   				IF NOT TailCurlSinStep THEN	
						
							hot_time_ton.IN:=TRUE;
							IF NOT arrCyCtrl[arrCyNo.CylinderName.PoleHotCutterCy].Cmd.bON AND NOT  arrCyCtrl[arrCyNo.CylinderName.PoleHotCutterCy].Status.ONState AND NOT hot_time_ton.Q THEN
								Mach_Control.WJ_b.HotCut:=TRUE;//启动热切
							END_IF
							
							IF hot_time_ton.Q THEN
							arrCyCtrl[arrCyNo.CylinderName.PoleHotCutterCy].Cmd.bON:=TRUE;//隔膜热切升降气缸伸出
							END_IF
							
							IF arrCyCtrl[arrCyNo.CylinderName.PoleHotCutterCy].Status.ONState  THEN
									Mach_Control.WJ_b.HotCut:=FALSE;//启动热切
									WJ_TON[1].IN:=FALSE;
									hot_time_ton.IN:=FALSE;
									TailCurlStep3:=205;	
								IF Mach_Control.WJ_b.SinStepMode THEN//尾卷单步模式
									TailCurlSinStep:=TRUE;
								ELSE
									TailCurlSinStep:=FALSE;
								END_IF								
							END_IF	
					END_IF
					


		305:
		
						
			SLCurlingneedleLine_TON.IN:=arrCyCtrl[arrCyNo.CylinderName.CurlingSplintCy_L].Status.OFFState AND arrCyCtrl[arrCyNo.CylinderName.CurlingSplintCy_S].Status.OFFState ;
				arrCyCtrl[arrCyNo.CylinderName.CurlingSplintCy_L].Cmd.bOFF:=TRUE;//尾卷长卷针张开
				arrCyCtrl[arrCyNo.CylinderName.CurlingSplintCy_S].Cmd.bOFF:=TRUE;//尾卷短卷针张开
				//arrCyCtrl[arrCyNo.CylinderName.CurlingSplintCy_S_1].Cmd.bON:=TRUE;//尾卷短卷针泄压关闭
				IF 	arrAxisCtrl[AxiseNo.AxisName.LCurlingneedleWhirling].Status.Homed AND arrAxisCtrl[AxiseNo.AxisName.LCurlingneedleWhirling].Status.NoMoving THEN
					IF arrAxisCtrl[AxiseNo.AxisName.LCurlingneedleWhirling].Cmd.arrbRealPoint[1] THEN
						arrAxisCtrl[AxiseNo.AxisName.LCurlingneedleWhirling].Cmd.iGoSetPos:=0;
					ELSE
						arrAxisCtrl[AxiseNo.AxisName.LCurlingneedleWhirling].Cmd.iGoSetPos:=1;//长卷针旋转至初始位
					END_IF
				END_IF										
				IF 	arrAxisCtrl[AxiseNo.AxisName.SCurlingneedleWhirling].Status.Homed AND arrAxisCtrl[AxiseNo.AxisName.SCurlingneedleWhirling].Status.NoMoving THEN
					IF arrAxisCtrl[AxiseNo.AxisName.SCurlingneedleWhirling].Cmd.arrbRealPoint[1] THEN
						arrAxisCtrl[AxiseNo.AxisName.SCurlingneedleWhirling].Cmd.iGoSetPos:=0;
					ELSE
						arrAxisCtrl[AxiseNo.AxisName.SCurlingneedleWhirling].Cmd.iGoSetPos:=1;//短卷针旋转至初始位
					END_IF
				END_IF
				IF 	 arrAxisCtrl[AxiseNo.AxisName.LCurlingneedleWhirling].Status.Moving AND arrAxisCtrl[AxiseNo.AxisName.SCurlingneedleWhirling].Status.Moving AND
					arrCyCtrl[arrCyNo.CylinderName.CurlingSplintCy_L].Status.OFFState AND arrCyCtrl[arrCyNo.CylinderName.CurlingSplintCy_S].Status.OFFState THEN														
					TailCurlStep3:=310;
				END_IF	
						

		1120:
	   				IF NOT TailCurlSinStep THEN	
						
							hot_time_ton.IN:=TRUE;
							IF NOT arrCyCtrl[arrCyNo.CylinderName.PoleHotCutterCy].Cmd.bON AND NOT  arrCyCtrl[arrCyNo.CylinderName.PoleHotCutterCy].Status.ONState AND NOT hot_time_ton.Q THEN
								Mach_Control.WJ_b.HotCut:=TRUE;//启动热切
							END_IF
							
							IF hot_time_ton.Q THEN
							arrCyCtrl[arrCyNo.CylinderName.PoleHotCutterCy].Cmd.bON:=TRUE;//隔膜热切升降气缸伸出
							END_IF
							
							IF arrCyCtrl[arrCyNo.CylinderName.PoleHotCutterCy].Status.ONState  THEN
									Mach_Control.WJ_b.HotCut:=FALSE;//启动热切
									WJ_TON[1].IN:=FALSE;
									hot_time_ton.IN:=FALSE;
									TailCurlStep3:=1140;	
								IF Mach_Control.WJ_b.SinStepMode THEN//尾卷单步模式
									TailCurlSinStep:=TRUE;
								ELSE
									TailCurlSinStep:=FALSE;
								END_IF								
							END_IF	
					END_IF			
				
				
				
END_CASE

 CASE TailCurlStep6 OF
10:
	IF (arrAxisCtrl[AxiseNo.AxisName.TailCurlSEPTALine].Status.fActPos<=(arrAxisPar[AxiseNo.AxisName.TailCurlSEPTALine].arrTargetPoint[1]+1)) OR Mach_Control.WJ_b.TailCurlDone  THEN
						 Mach_Control.DT_b.OffloadDone:=TRUE;
						 TailCurlStep6:=20;
					END_IF
					
20:
	TailCurlStep6:=666;

END_CASE 













//尾卷拉膜耦合放卷虚轴			
tailCult_GearInMultiMaster(
	Master1:=arrAxis[AxiseNo.AxisName.TailCurlRetracting] , 
	Master2:=arrAxis[AxiseNo.AxisName.TailCurlLine]  , 
	Master3:=arrAxis[AxiseNo.VirAxisName.VirDriver]  , 
	Master4:=arrAxis[AxiseNo.VirAxisName.VirDriver]  , 
	Slave:=arrAxis[AxiseNo.VirAxisName.VirDriver], 
	Enable:=tailCult_GearInMultiMaster.Enable , 
	GearRatio1:=-1 , 
	GearRatio2:=-1 , 
	GearRatio3:=0 , 
	GearRatio4:=0, 
	Acceleration:= , 
	Deceleration:= , 
	Jerk:= , 
	BufferMode:= , 
	Options:= , 
	InGear=> , 
	Busy=> , 
	Active=> , 
	CommandAborted=> , 
	Error=> , 
	ErrorID=> );				
tailCult_GearInMultiMaster.Error;
tailCult_GearInMultiMaster.Busy;	

//放卷虚轴解除耦合
fTailCurl_TRIG(CLK:=tailCult_GearInMultiMaster.Enable , Q=> );
tailCurl_CamOut(
	Slave:=arrAxis[AxiseNo.VirAxisName.VirDriver]  , 
	Execute:=fTailCurl_TRIG.Q , 
	Options:= , 
	Done=> , 
	Busy=> , 
	Error=> , 
	ErrorID=> );	
	
	
		
//夹电芯平移轴与夹隔膜平移轴电子齿轮耦合
	
	tailCurl_GearIn(
	Reset:=        stSysState.bReset  , 
	fratio1:= 1, 
	bError=> , 
	bReady=> , 
	InGear=> , 
	bEnable:=     tailCurlGearInEnable    , 
	master:=       arrAxis[AxiseNo.AxisName.TailCurlLine]  , 
	slave1:=        arrAxis[AxiseNo.AxisName.TailCurlSEPTALine], );
	tailCurl_GearIn.InGear;
	tailCurl_GearIn.bError;
	tailCurl_GearIn.bReady;
	
	
//夹电芯平移轴与夹隔膜平移轴电子齿轮耦合--取料
tailCurl_GearIn1.fratio1:=(arrAxisPar[AxiseNo.AxisName.TailCurlSEPTALine].arrTargetPoint[2]-arrAxisPar[AxiseNo.AxisName.TailCurlSEPTALine].arrTargetPoint[1])/(arrAxisPar[AxiseNo.AxisName.TailCurlLine].arrTargetPoint[2]-arrAxisPar[AxiseNo.AxisName.TailCurlLine].arrTargetPoint[11]);;
tailCurl_GearIn1(
	Reset:=        stSysState.bReset  , 
	fratio1:= , 
	bError=> , 
	bReady=> , 
	InGear=> , 
	bEnable:=     tailCurlGearInEnable1    , 
	master:=       arrAxis[AxiseNo.AxisName.TailCurlLine]  , 
	slave1:=        arrAxis[AxiseNo.AxisName.TailCurlSEPTALine], );
	tailCurl_GearIn1.InGear;
	tailCurl_GearIn1.bError;
	tailCurl_GearIn1.bReady;
		
	
	
//尾卷夹电芯伸缩取料齿轮耦合
tailRetGearIn.fratio1:=(arrAxisPar[AxiseNo.AxisName.TailCurlRetracting].arrTargetPoint[2]-arrAxisPar[AxiseNo.AxisName.TailCurlRetracting].arrTargetPoint[1])/(arrAxisPar[AxiseNo.AxisName.TailCurlLine].arrTargetPoint[2]-arrAxisPar[AxiseNo.AxisName.TailCurlLine].arrTargetPoint[11]);
	tailRetGearIn(
	Reset:=        stSysState.bReset  , 
	fratio1:= , 
	bError=> , 
	bReady=> , 
	InGear=> , 
	bEnable:=     tailRetGearInEnable    , 
	master:=       arrAxis[AxiseNo.AxisName.TailCurlLine]  , 
	slave1:=        arrAxis[AxiseNo.AxisName.TailCurlRetracting], );
	tailRetGearIn.InGear;
	tailRetGearIn.bError;
	tailRetGearIn.bReady;
	


//长、短卷针平移电子齿轮耦合  CurlingneedleLine    FB_GearInDyn
	CurlingneedleLine_GearIn(
	Reset:=        stSysState.bReset  , 
	fratio1:= -1, 
	bError=> , 
	bReady=> , 
	InGear=> , 
	bEnable:=     CurlingneedleLineEnable    , 
	master:=       arrAxis[AxiseNo.AxisName.LCurlingneedleLine]  , 
	slave1:=        arrAxis[AxiseNo.AxisName.SCurlingneedleLine], );
	
	CurlingneedleLine_GearIn.InGear;
	CurlingneedleLine_GearIn.bError;
	CurlingneedleLine_GearIn.bReady;
END_ACTION

ACTION TailCurl_Auto2:
//判断尾卷是否有轴在耕合中
IF arrAxisCtrl[AxiseNo.AxisName.TailCurlSEPTALine].Status.Coupled OR arrAxisCtrl[AxiseNo.AxisName.TailCurlSEPTAUpDown].Status.Coupled OR  
	arrAxisCtrl[AxiseNo.AxisName.LCurlingneedleWhirling].Status.Coupled OR arrAxisCtrl[AxiseNo.AxisName.SCurlingneedleWhirling].Status.Coupled THEN
	TailCurlCoupling:=TRUE;//尾卷轴耦合中
ELSE
	TailCurlCoupling:=FALSE;
END_IF



IF Mach_Control.U.WJ_iMode=1  THEN//在自动状态下
//尾卷电芯自动
		CASE TailCurlStep4 OF
			0://判断尾卷是否启动
					IF TailCurlStart THEN
						TailCurlStart:=FALSE;//复位尾卷启动
						Mach_Control.WJ_b.TailCurlDone:=FALSE;	//尾卷完成
						arrAxisCtrl[AxiseNo.VirAxisName.VirTailCurl].Cmd.bMoveAbs:=FALSE;//主轴启动
						TailCurlStep4:=10;
					END_IF
			10://尾卷凸轮耦合，判断尾卷主轴是停止、当前位置是否为0
				 	IF arrAxis[AxiseNo.VirAxisName.VirTailCurl].Status.NotMoving AND ABS(arrAxis[AxiseNo.VirAxisName.VirTailCurl].NcToPlc.ActPos)<=0.1 AND NOT TailCurlCoupling THEN
						TailCurlStep4:=30;
					ELSE
						TailCurlStep0:=50;
						TailCurlStep4:=20;			
					END_IF		
			20://等待主轴停止并且清零完成
					IF TailCurlStep0=6666 THEN
						TailCurlStep4:=30;	
					END_IF
					
			30://凸轮耦合
					fbCamInEndWindX.bCamInExecute:=TRUE;//夹膜平移轴凸轮耦合
					fbCamInEndWindY.bCamInExecute:=TRUE;//夹膜升降轴凸轮耦合
					tailCurl1_GearIn.Execute:=TRUE;//短卷针齿轮耦合
					tailCurl2_GearIn.Execute:=TRUE;//长卷针齿轮耦合
					IF arrAxisCtrl[AxiseNo.AxisName.TailCurlSEPTALine].Status.Coupled AND  arrAxisCtrl[AxiseNo.AxisName.TailCurlSEPTAUpDown].Status.Coupled AND   
						arrAxisCtrl[AxiseNo.AxisName.LCurlingneedleWhirling].Status.Coupled AND arrAxisCtrl[AxiseNo.AxisName.SCurlingneedleWhirling].Status.Coupled THEN
						TailCurlStep4:=40;	
					END_IF
			40://主轴启动
					arrAxisCtrl[AxiseNo.VirAxisName.VirTailCurl].Cmd.bDynamitcsParSel:=2;
					arrAxisCtrl[AxiseNo.VirAxisName.VirTailCurl].Cmd.fPositon_of_Abs:=359.5*Par.stWJ_date.SumNo;
					arrAxisPar[AxiseNo.VirAxisName.VirTailCurl].fTagatTime:=Par.stWJ_date.CoeSpeed;
					arrAxisCtrl[AxiseNo.VirAxisName.VirTailCurl].Cmd.bMoveAbs:=TRUE;
					TailCurlStep4:=50;	
					TailCurlStep5:=10;//夹膜平移超限凸轮解除耦合
			50://	解除夹隔平移、夹隔升降凸轮耦合	
				IF NOT TailCurlSinStep THEN
					IF arrAxisCtrl[AxiseNo.VirAxisName.VirTailCurl].Status.fSetPos=359.5*Par.stWJ_date.SumNo AND arrAxisCtrl[AxiseNo.VirAxisName.VirTailCurl].Status.NoMoving AND 
                       TailCurlStep5=6666 THEN				
						fbCamInEndWindX.bCamInExecute:=FALSE;//夹膜平移轴凸轮耦合					
						fbCamInEndWindY.bCamInExecute:=FALSE;//夹膜升降轴凸轮耦合
						IF NOT arrAxisCtrl[AxiseNo.AxisName.TailCurlSEPTALine].Status.Coupled AND NOT arrAxisCtrl[AxiseNo.AxisName.TailCurlSEPTAUpDown].Status.Coupled THEN
								IF Mach_Control.WJ_b.SinStepMode THEN//尾卷单步模式
									TailCurlSinStep:=TRUE;
								ELSE
									TailCurlSinStep:=FALSE;
								END_IF
							TailCurlStep0 :=50;
							TailCurlStep4:=60;	
						END_IF
					END_IF
				END_IF
			60:
				IF TailCurlStep0=6666 THEN
					Mach_Control.WJ_b.TailCurlDone	:=TRUE;	//尾卷完成
					TailCurlStep4:=0;
				END_IF
			(*60://压隔膜平移气缸伸出、压隔膜平移升降气缸	
				arrCyCtrl[arrCyNo.CylinderName.PoleSplintCy_D].Cmd.bOFF:=TRUE;//尾卷夹隔膜下夹板收回位
				//arrCyCtrl[arrCyNo.CylinderName.TailCurlLineCy].Cmd.bON:=TRUE;//尾卷压轮平移气缸伸出
				//IF arrCyCtrl[arrCyNo.CylinderName.TailCurlLineCy].Status.ONState THEN
					//arrCyCtrl[arrCyNo.CylinderName.TailCurlUpdownCy].Cmd.bON:=TRUE;//尾卷压轮升降气缸下降
					//IF arrCyCtrl[arrCyNo.CylinderName.TailCurlUpdownCy].Status.ONState THEN
						TailCurlStep4:=70;
				//	END_IF				
				//END_IF
			70://夹隔膜平移至初始位，夹隔膜升降至初始位
				
				IF arrCyCtrl[arrCyNo.CylinderName.PoleSplintCy_D].Status.OFFState THEN
						IF 	 arrAxisCtrl[AxiseNo.AxisName.TailCurlSEPTALine].Status.Homed AND arrAxisCtrl[AxiseNo.AxisName.TailCurlSEPTALine].Status.NoMoving THEN
							IF arrAxisCtrl[AxiseNo.AxisName.TailCurlSEPTALine].Cmd.arrbRealPoint[1] THEN
								arrAxisCtrl[AxiseNo.AxisName.TailCurlSEPTALine].Cmd.iGoSetPos:=0;
							ELSE
								arrAxisCtrl[AxiseNo.AxisName.TailCurlSEPTALine].Cmd.iGoSetPos:=1;//尾卷夹隔膜平移初始位
							END_IF
						END_IF	
						IF 	 arrAxisCtrl[AxiseNo.AxisName.TailCurlSEPTAUpDown].Status.Homed AND arrAxisCtrl[AxiseNo.AxisName.TailCurlSEPTAUpDown].Status.NoMoving THEN
							IF arrAxisCtrl[AxiseNo.AxisName.TailCurlSEPTAUpDown].Cmd.arrbRealPoint[1] THEN
								arrAxisCtrl[AxiseNo.AxisName.TailCurlSEPTAUpDown].Cmd.iGoSetPos:=0;
							ELSE
								arrAxisCtrl[AxiseNo.AxisName.TailCurlSEPTAUpDown].Cmd.iGoSetPos:=1;//尾卷夹隔膜升降初始位
							END_IF
						END_IF
						IF 	arrAxisCtrl[AxiseNo.AxisName.TailCurlSEPTALine].Cmd.arrbRealPoint[1] AND  arrAxisCtrl[AxiseNo.AxisName.TailCurlSEPTAUpDown].Cmd.arrbRealPoint[1]  THEN
							TailCurlStep0 :=50;
							Mach_Control.WJ_b.TailCurlDone	:=TRUE;	//尾卷完成
							TailCurlStep4:=0;
						END_IF	
				END_IF		
			80://启动主轴
					arrAxisCtrl[AxiseNo.VirAxisName.VirTailCurl].Cmd.bDynamitcsParSel:=2;
					arrAxisCtrl[AxiseNo.VirAxisName.VirTailCurl].Cmd.fPositon_of_Abs:=540;
					arrAxisPar[AxiseNo.VirAxisName.VirTailCurl].fTagatTime:=20;
					arrAxisCtrl[AxiseNo.VirAxisName.VirTailCurl].Cmd.bMoveAbs:=TRUE;	
					TailCurlStep4:=90;
			90://判断主轴运动是否完成
					IF arrAxisCtrl[AxiseNo.VirAxisName.VirTailCurl].Status.fSetPos=540 AND arrAxisCtrl[AxiseNo.VirAxisName.VirTailCurl].Status.NoMoving THEN
							tailCurl1_GearIn.Execute:=FALSE;//短卷针齿轮耦合
							tailCurl2_GearIn.Execute:=FALSE;//长卷针齿轮耦合
							IF NOT arrAxisCtrl[AxiseNo.AxisName.LCurlingneedleWhirling].Status.Coupled AND NOT arrAxisCtrl[AxiseNo.AxisName.SCurlingneedleWhirling].Status.Coupled  THEN
								Mach_Control.WJ_b.TailCurlDone	:=TRUE;	//尾卷完成
								TailCurlStep0 :=50;
								TailCurlStep4:=0;	
							END_IF
					END_IF	*)		
		END_CASE
		
//尾卷主轴停止，当前位置清零
		CASE TailCurlStep0 OF
				50:
					TailCurlStep0:=100;
					
				100://判断主轴是否在运动中
					IF NOT TailCurlSinStep THEN
						IF arrAxis[AxiseNo.VirAxisName.VirTailCurl].Status.NotMoving  THEN
							arrAxisCtrl[AxiseNo.VirAxisName.VirTailCurl].Cmd.bStop:=FALSE;
							TailCurlStep0:=110;
								IF Mach_Control.WJ_b.SinStepMode THEN//尾卷单步模式
												TailCurlSinStep:=TRUE;
											ELSE
												TailCurlSinStep:=FALSE;
											END_IF
						ELSE
							arrAxisCtrl[AxiseNo.VirAxisName.VirTailCurl].Cmd.bStop:=TRUE;//尾卷主轴停止
						END_IF
						END_IF
				110://判断尾卷轴是否在耦合中
					IF NOT TailCurlSinStep THEN
						IF TailCurlCoupling  THEN
								TailCurlStep0:=120;
										IF Mach_Control.WJ_b.SinStepMode THEN//尾卷单步模式
												TailCurlSinStep:=TRUE;
											ELSE
												TailCurlSinStep:=FALSE;
											END_IF
						ELSE
								TailCurlStep0:=130;
										IF Mach_Control.WJ_b.SinStepMode THEN//尾卷单步模式
												TailCurlSinStep:=TRUE;
											ELSE
												TailCurlSinStep:=FALSE;
											END_IF
						END_IF
						END_IF
				120://尾卷凸轮解除耦合
						fbCamInEndWindX.bCamInExecute:=FALSE;
						fbCamInEndWindY.bCamInExecute:=FALSE;
						tailCurl1_GearIn.Execute:=FALSE;//短卷针齿轮耦合
						tailCurl2_GearIn.Execute:=FALSE;//长卷针齿轮耦合
						IF  NOT TailCurlCoupling THEN
							TailCurlStep0:=125;
						END_IF
						
				125:
					IF NOT TailCurlSinStep THEN
						arrAxisCtrl[AxiseNo.AxisName.TailCurlSEPTALine].Cmd.bStop:=TRUE;
						IF arrAxisCtrl[AxiseNo.AxisName.TailCurlSEPTALine].Status.NoMoving AND NOT arrAxisCtrl[AxiseNo.AxisName.TailCurlSEPTALine].Status.Coupled THEN
							
							IF Mach_Control.WJ_b.SinStepMode THEN//尾卷单步模式
								TailCurlSinStep:=TRUE;
							ELSE
								TailCurlSinStep:=FALSE;
							END_IF	
							arrAxisCtrl[AxiseNo.AxisName.TailCurlSEPTALine].Cmd.bStop:=FALSE;
							TailCurlStep0:=130;
						END_IF
					END_IF
				130://主轴当前位置清零
						IF NOT arrAxisCtrl[AxiseNo.AxisName.TailCurlSEPTALine].Status.Coupled AND 
							NOT arrAxisCtrl[AxiseNo.AxisName.TailCurlSEPTAUpDown].Status.Coupled THEN
									arrAxisCtrl[AxiseNo.VirAxisName.VirTailCurl].Cmd.fSetPos:=0;
									arrAxisCtrl[AxiseNo.VirAxisName.VirTailCurl].Cmd.bSetPos:=TRUE;	
									TailCurlStep0:=140;
						END_IF
				140://判断主轴清零是否完成
						//IF arrAxis[AxiseNo.VirAxisName.VirTailCurl].Status.NotMoving  AND arrAxis[AxiseNo.VirAxisName.VirTailCurl].NcToPlc.SetPos=0 THEN		
							TailCurlStep0:=150;
						//END_IF
						
						
				150:
					arrAxisCtrl[AxiseNo.VirAxisName.VirTailCurl].Cmd.bEnable:=FALSE;
					WJ_TON[3](IN:=NOT arrAxisCtrl[AxiseNo.VirAxisName.VirTailCurl].Cmd.bEnable, PT:=T#20MS, Q=> , ET=> );	
					IF WJ_TON[3].Q  THEN
						arrAxisCtrl[AxiseNo.VirAxisName.VirTailCurl].Cmd.bSetPos:=FALSE;
						arrAxisCtrl[AxiseNo.VirAxisName.VirTailCurl].Cmd.bStop:=FALSE;	
						WJ_TON[3](IN:=FALSE);	
						TailCurlStep0:=160;
					END_IF
				160:
					WJ_TON[4](IN:=FALSE);	
					arrAxisCtrl[AxiseNo.VirAxisName.VirTailCurl].Cmd.bEnable:=TRUE;	
					TailCurlStep0:=170;
				170:
					arrAxisCtrl[AxiseNo.VirAxisName.VirTailCurl].Cmd.bReset:=TRUE;
					WJ_TON[4](IN:=TRUE, PT:=T#20MS, Q=> , ET=> );	
					IF WJ_TON[4].Q THEN
						WJ_TON[4](IN:=FALSE);	
						TailCurlStep0:=180;
					END_IF
				180:	
					arrAxisCtrl[AxiseNo.VirAxisName.VirTailCurl].Cmd.bReset:=FALSE;	
					TailCurlStep0:=190;
						
				190:		
					IF arrAxis[AxiseNo.VirAxisName.VirTailCurl].Status.NotMoving  AND arrAxis[AxiseNo.VirAxisName.VirTailCurl].NcToPlc.SetPos=0 
						AND arrAxisCtrl[AxiseNo.VirAxisName.VirTailCurl].Cmd.bEnable THEN
						TailCurlStep0:=6666;
					END_IF		
						
		END_CASE
END_IF


CASE  TailCurlStep5 OF
10:
	IF arrAxisCtrl[AxiseNo.VirAxisName.VirTailCurl].Status.fActPos>0  AND arrAxisCtrl[AxiseNo.AxisName.TailCurlSEPTALine].Status.fSetPos<=(par.stWJ_date.WJ_PoistCamOut+2 ) 
		AND arrAxisCtrl[AxiseNo.VirAxisName.VirTailCurl].Status.fActPos<=357 THEN//解耦
		fbCamInEndWindX.bGearOutMode:=TRUE;//夹膜平移轴凸轮耦合
		fbCamInEndWindX.bCamInExecute:=FALSE;//夹膜平移轴凸轮耦合
		
		IF NOT fbCamInEndWindX.bCamInExecute THEN
			TailCurlStep5:=100;
		END_IF
	ELSIF arrAxisCtrl[AxiseNo.VirAxisName.VirTailCurl].Status.fActPos>357 AND arrAxisCtrl[AxiseNo.AxisName.TailCurlSEPTALine].Status.fSetPos>=par.stWJ_date.WJ_PoistCamOut THEN//不解耦
		TailCurlStep5:=6666;
	END_IF
	
100:
	IF NOT  fbCamInEndWindX.bCamInExecute AND NOT arrAxisCtrl[AxiseNo.AxisName.TailCurlSEPTALine].Status.Coupled AND NOT fbCamInEndWindX.bInSync  THEN
		TailCurlStep5:=200;
	END_IF
200://高速定位停止
	arrAxisCtrl[AxiseNo.AxisName.TailCurlSEPTALine].Cmd.bDynamitcsParSel:=2;
	arrAxisCtrl[AxiseNo.AxisName.TailCurlSEPTALine].Cmd.fPositon_of_Abs:=par.stWJ_date.WJ_PoistCamOut-1;
	arrAxisPar[AxiseNo.AxisName.TailCurlSEPTALine].fTagatTime:= 0.02;//3.33333/arrAxisPar[AxiseNo.AxisName.TailCurlSEPTALine].fVelocity_of_Abs+0.01 
	arrAxisCtrl[AxiseNo.AxisName.TailCurlSEPTALine].Cmd.bMoveAbs:=TRUE;
	TailCurlStep5:=300;
300:
	IF ABS(arrAxisCtrl[AxiseNo.AxisName.TailCurlSEPTALine].Status.fActPos+1-par.stWJ_date.WJ_PoistCamOut)<=0.5 AND NOT arrAxisCtrl[AxiseNo.AxisName.TailCurlSEPTALine].Cmd.bMoveAbs
	AND arrAxisCtrl[AxiseNo.AxisName.TailCurlSEPTALine].Status.NoMoving THEN
		arrAxisCtrl[AxiseNo.AxisName.TailCurlSEPTALine].Cmd.bMoveAbs:=FALSE;
		TailCurlStep5:=400;
	END_IF
400:
	arrAxisCtrl[AxiseNo.AxisName.TailCurlSEPTALine].Cmd.bDynamitcsParSel:=1;
	fbCamInEndWindX.bGearOutMode:=FALSE;//夹膜平移轴凸轮耦合
	IF arrAxisCtrl[AxiseNo.AxisName.TailCurlSEPTALine].Cmd.bDynamitcsParSel=1 THEN
		TailCurlStep5:=6666;
	END_IF
END_CASE

(*
CASE  TailCurlStep5 OF
			10:
					IF 	 arrAxisCtrl[AxiseNo.VirAxisName.VirTailCurl].Status.fActPos>0  AND arrAxisCtrl[AxiseNo.AxisName.TailCurlSEPTALine].Status.fSetPos<=par.stWJ_date.WJ_PoistCamOut   THEN
							fbCamInEndWindX.bCamInExecute:=FALSE;//夹膜平移轴凸轮耦合
							//arrAxisCtrl[AxiseNo.AxisName.SEPTATLine].Cmd.bStop:=TRUE;
					END_IF
					IF NOT fbCamInEndWindX.bCamInExecute THEN
						TailCurlStep5:=6666;
					END_IF
END_CASE
*)
(**************************************夹膜平移正常解耦位计算******************************************************)
arrAxisPar[AxiseNo.AxisName.TailCurlSEPTALine].arrTargetPoint[4]:=arrAxisPar[AxiseNo.AxisName.TailCurlSEPTALine].arrTargetPoint[2]
								-(arrAxisPar[AxiseNo.AxisName.TailCurlLine].arrTargetPoint[7]-arrAxisPar[AxiseNo.AxisName.TailCurlLine].arrTargetPoint[4])
								-(fbRoll_New.AxisXmm*2);
END_ACTION

ACTION TailCurl_Condition:
//尾卷夹电芯平移轴移动至初始位置的安全件件
(*
IF  arrAxis[AxiseNo.AxisName.TailCurlWhirling].Status.Homed AND arrAxisCtrl[AxiseNo.AxisName.TailCurlWhirling].Status.NoMoving AND
	(arrAxisCtrl[AxiseNo.AxisName.TailCurlWhirling].Cmd.arrbRealPoint[1] OR arrAxisCtrl[AxiseNo.AxisName.TailCurlWhirling].Cmd.arrbRealPoint[2]) AND	
	arrAxisCtrl[AxiseNo.AxisName.LCurlingneedleLine].Status.Homed AND arrAxisCtrl[AxiseNo.AxisName.LCurlingneedleLine].Status.NoMoving AND arrAxisCtrl[AxiseNo.AxisName.LCurlingneedleLine].Cmd.arrbRealPoint[1] AND 
	arrAxisCtrl[AxiseNo.AxisName.SCurlingneedleLine].Status.Homed AND arrAxisCtrl[AxiseNo.AxisName.SCurlingneedleLine].Status.NoMoving AND arrAxisCtrl[AxiseNo.AxisName.SCurlingneedleLine].Cmd.arrbRealPoint[1]  
OR Mach_Control.WJ_b.AxisConditionEN THEN
	arrAxisCtrl[AxiseNo.AxisName.TailCurlLine].Cmd.GoPoint_Condition[1]:=TRUE;
ELSE
	arrAxisCtrl[AxiseNo.AxisName.TailCurlLine].Cmd.GoPoint_Condition[1]:=FALSE;
END_IF

//尾卷夹隔膜轴移动至取电芯位的安全条件
IF arrAxisCtrl[AxiseNo.AxisName.CaDTCarryingLine].Status.Homed AND arrAxisCtrl[AxiseNo.AxisName.CaDTCarryingLine].Status.NoMoving AND arrAxisCtrl[AxiseNo.AxisName.CaDTCarryingLine].Cmd.arrbRealPoint[1] 
OR Mach_Control.WJ_b.AxisConditionEN THEN	
	arrAxisCtrl[AxiseNo.AxisName.TailCurlSEPTALine].Cmd.GoPoint_Condition[2]:=TRUE;
ELSE
	arrAxisCtrl[AxiseNo.AxisName.TailCurlSEPTALine].Cmd.GoPoint_Condition[2]:=FALSE;	
END_IF
*)

/////////////////////////////////////////////////////////////
/////////////////////////////////////////////////////////
////////////////////////////////////////////电机条件
//尾卷夹电芯平移 
IF  Mach_Control.U.WJ_iMode=3 AND 
	arrAxisCtrl[AxiseNo.AxisName.LCurlingneedleLine].Status.fActPos<=arrAxisPar[AxiseNo.AxisName.LCurlingneedleLine].arrTargetPoint[1]+1 AND arrAxisCtrl[AxiseNo.AxisName.LCurlingneedleLine].Status.Homed  AND
	arrAxisCtrl[AxiseNo.AxisName.SCurlingneedleLine].Status.fActPos <=arrAxisPar[AxiseNo.AxisName.SCurlingneedleLine] .arrTargetPoint[1]+1 AND arrAxisCtrl[AxiseNo.AxisName.SCurlingneedleLine].Status.Homed AND 
	(arrAxisCtrl[AxiseNo.AxisName.TailCurlWhirling].Status.fActPos<=arrAxisPar[AxiseNo.AxisName.TailCurlWhirling].arrTargetPoint[1]+1 AND
	arrAxisCtrl[AxiseNo.AxisName.TailCurlWhirling].Status.fActPos>=arrAxisPar[AxiseNo.AxisName.TailCurlWhirling].arrTargetPoint[1]-1	) OR 
	(arrAxisCtrl[AxiseNo.AxisName.TailCurlWhirling].Status.fActPos<=arrAxisPar[AxiseNo.AxisName.TailCurlWhirling].arrTargetPoint[2]+1 AND
	arrAxisCtrl[AxiseNo.AxisName.TailCurlWhirling].Status.fActPos>=arrAxisPar[AxiseNo.AxisName.TailCurlWhirling].arrTargetPoint[2]-1	) 
    OR Mach_Control.WJ_b.AxisConditionEN THEN
	arrAxisCtrl[AxiseNo.AxisName.TailCurlLine].Cmd.Home_Condition:=TRUE;
ELSE
	arrAxisCtrl[AxiseNo.AxisName.TailCurlLine].Cmd.Home_Condition:=FALSE;	
END_IF

IF Mach_Control.U.WJ_iMode=3 AND
	arrAxisCtrl[AxiseNo.AxisName.LCurlingneedleLine].Status.fActPos<=arrAxisPar[AxiseNo.AxisName.LCurlingneedleLine].arrTargetPoint[1]+1 AND arrAxisCtrl[AxiseNo.AxisName.LCurlingneedleLine].Status.Homed  AND
	arrAxisCtrl[AxiseNo.AxisName.SCurlingneedleLine].Status.fActPos <=arrAxisPar[AxiseNo.AxisName.SCurlingneedleLine] .arrTargetPoint[1]+1 AND arrAxisCtrl[AxiseNo.AxisName.SCurlingneedleLine].Status.Homed 
 THEN
   arrAxisCtrl[AxiseNo.AxisName.TailCurlLine].Cmd.JogP_Condition:=TRUE;
   arrAxisCtrl[AxiseNo.AxisName.TailCurlLine].Cmd.JogN_Condition:=TRUE;
   ELSE 
   arrAxisCtrl[AxiseNo.AxisName.TailCurlLine].Cmd.JogP_Condition:=FALSE;
   arrAxisCtrl[AxiseNo.AxisName.TailCurlLine].Cmd.JogN_Condition:=FALSE;
 END_IF

IF  Mach_Control.U.WJ_iMode=3 AND arrAxisCtrl[AxiseNo.AxisName.TailCurlLine].Status.Homed 
AND (arrAxisCtrl[AxiseNo.AxisName.TailCurlWhirling].Cmd.arrbRealPoint[1] OR  arrAxisCtrl[AxiseNo.AxisName.TailCurlWhirling].Cmd.arrbRealPoint[2]) AND
arrAxisCtrl[AxiseNo.AxisName.LCurlingneedleLine].Status.fActPos<=arrAxisPar[AxiseNo.AxisName.LCurlingneedleLine].arrTargetPoint[1]+1 AND arrAxisCtrl[AxiseNo.AxisName.LCurlingneedleLine].Status.Homed  AND
arrAxisCtrl[AxiseNo.AxisName.SCurlingneedleLine].Status.fActPos <=arrAxisPar[AxiseNo.AxisName.SCurlingneedleLine] .arrTargetPoint[1]+1 AND arrAxisCtrl[AxiseNo.AxisName.SCurlingneedleLine].Status.Homed 
OR Mach_Control.WJ_b.AxisConditionEN THEN
	arrAxisCtrl[AxiseNo.AxisName.TailCurlLine].Cmd.GoPoint_Condition[1]:=TRUE;
ELSE
	arrAxisCtrl[AxiseNo.AxisName.TailCurlLine].Cmd.GoPoint_Condition[1]:=FALSE;	
END_IF

IF  Mach_Control.U.WJ_iMode=3 AND arrAxisCtrl[AxiseNo.AxisName.TailCurlLine].Status.Homed 
AND (arrAxisCtrl[AxiseNo.AxisName.TailCurlWhirling].Cmd.arrbRealPoint[1]
AND NOT arrAxisCtrl[AxiseNo.AxisName.TailCurlWhirling].Cmd.arrbRealPoint[2]
AND arrAxisCtrl[AxiseNo.AxisName.TailCurlSEPTAUpDown].Cmd.arrbRealPoint[1]  
AND  arrCyCtrl[arrCyNo.CylinderName.PoleHotCutterCy].Status.OFFState
AND  arrAxisCtrl[AxiseNo.AxisName.LCurlingneedleLine].Status.fActPos<=arrAxisPar[AxiseNo.AxisName.LCurlingneedleLine].arrTargetPoint[1]+1 AND arrAxisCtrl[AxiseNo.AxisName.LCurlingneedleLine].Status.Homed  
AND arrAxisCtrl[AxiseNo.AxisName.SCurlingneedleLine].Status.fActPos <=arrAxisPar[AxiseNo.AxisName.SCurlingneedleLine] .arrTargetPoint[1]+1 AND arrAxisCtrl[AxiseNo.AxisName.SCurlingneedleLine].Status.Homed 
AND arrAxisCtrl[AxiseNo.AxisName.TailCurlUpDown].Cmd.arrbRealPoint[1] )
AND  arrCyCtrl[arrCyNo.CylinderName.TailCurlSplintCy].Io.DIOFFSwitch 
AND arrCyCtrl[arrCyNo.CylinderName.PoleSplintCy_D].Status.OFFState
AND arrAxisCtrl[AxiseNo.AxisName.TailCurlSEPTALine].Cmd.arrbRealPoint[2]
AND  arrAxisCtrl[AxiseNo.AxisName.SEPTATLine].Cmd.arrbRealPoint[1] 
  OR Mach_Control.WJ_b.AxisConditionEN THEN
	arrAxisCtrl[AxiseNo.AxisName.TailCurlLine].Cmd.GoPoint_Condition[2]:=TRUE;
ELSE
	arrAxisCtrl[AxiseNo.AxisName.TailCurlLine].Cmd.GoPoint_Condition[2]:=FALSE;	
END_IF

IF  Mach_Control.U.WJ_iMode=3 AND arrAxisCtrl[AxiseNo.AxisName.TailCurlLine].Status.Homed 
AND (arrAxisCtrl[AxiseNo.AxisName.TailCurlWhirling].Cmd.arrbRealPoint[1] 
AND NOT  arrAxisCtrl[AxiseNo.AxisName.TailCurlWhirling].Cmd.arrbRealPoint[2]) 
AND  arrAxisCtrl[AxiseNo.AxisName.LCurlingneedleLine].Status.fActPos<=arrAxisPar[AxiseNo.AxisName.LCurlingneedleLine].arrTargetPoint[1]+1 AND arrAxisCtrl[AxiseNo.AxisName.LCurlingneedleLine].Status.Homed  
AND  arrAxisCtrl[AxiseNo.AxisName.SCurlingneedleLine].Status.fActPos <=arrAxisPar[AxiseNo.AxisName.SCurlingneedleLine] .arrTargetPoint[1]+1 AND arrAxisCtrl[AxiseNo.AxisName.SCurlingneedleLine].Status.Homed 
OR Mach_Control.WJ_b.AxisConditionEN THEN
	arrAxisCtrl[AxiseNo.AxisName.TailCurlLine].Cmd.GoPoint_Condition[3]:=TRUE;
ELSE
	arrAxisCtrl[AxiseNo.AxisName.TailCurlLine].Cmd.GoPoint_Condition[3]:=FALSE;	
END_IF

IF  Mach_Control.U.WJ_iMode=3 AND arrAxisCtrl[AxiseNo.AxisName.TailCurlLine].Status.Homed 
AND arrAxisCtrl[AxiseNo.AxisName.TailCurlWhirling].Cmd.arrbRealPoint[1] 
AND arrAxisCtrl[AxiseNo.AxisName.LCurlingneedleLine].Status.fActPos<=arrAxisPar[AxiseNo.AxisName.LCurlingneedleLine].arrTargetPoint[1] +1
AND arrAxisCtrl[AxiseNo.AxisName.LCurlingneedleLine].Status.Homed  
AND arrAxisCtrl[AxiseNo.AxisName.SCurlingneedleLine].Status.fActPos <=arrAxisPar[AxiseNo.AxisName.SCurlingneedleLine] .arrTargetPoint[1]+1 
AND arrAxisCtrl[AxiseNo.AxisName.SCurlingneedleLine].Status.Homed 
OR Mach_Control.WJ_b.AxisConditionEN THEN
	arrAxisCtrl[AxiseNo.AxisName.TailCurlLine].Cmd.GoPoint_Condition[4]:=TRUE;
ELSE
	arrAxisCtrl[AxiseNo.AxisName.TailCurlLine].Cmd.GoPoint_Condition[4]:=FALSE;	
END_IF

IF  Mach_Control.U.WJ_iMode=3 AND arrAxisCtrl[AxiseNo.AxisName.TailCurlLine].Status.Homed  
AND arrAxisCtrl[AxiseNo.AxisName.TailCurlWhirling].Cmd.arrbRealPoint[1] 
AND arrAxisCtrl[AxiseNo.AxisName.LCurlingneedleLine].Status.fActPos<=arrAxisPar[AxiseNo.AxisName.LCurlingneedleLine].arrTargetPoint[1]+1 
AND arrAxisCtrl[AxiseNo.AxisName.LCurlingneedleLine].Status.Homed  
AND arrAxisCtrl[AxiseNo.AxisName.SCurlingneedleLine].Status.fActPos <=arrAxisPar[AxiseNo.AxisName.SCurlingneedleLine] .arrTargetPoint[1]+1 
AND arrAxisCtrl[AxiseNo.AxisName.SCurlingneedleLine].Status.Homed 
OR Mach_Control.WJ_b.AxisConditionEN THEN
	arrAxisCtrl[AxiseNo.AxisName.TailCurlLine].Cmd.GoPoint_Condition[5]:=TRUE;
ELSE
	arrAxisCtrl[AxiseNo.AxisName.TailCurlLine].Cmd.GoPoint_Condition[5]:=FALSE;	
END_IF

IF  Mach_Control.U.WJ_iMode=3 AND arrAxisCtrl[AxiseNo.AxisName.TailCurlLine].Status.Homed 
AND arrAxisCtrl[AxiseNo.AxisName.TailCurlWhirling].Cmd.arrbRealPoint[2] 
AND arrAxisCtrl[AxiseNo.AxisName.LCurlingneedleLine].Status.fActPos<=arrAxisPar[AxiseNo.AxisName.LCurlingneedleLine].arrTargetPoint[1]+1 
AND arrAxisCtrl[AxiseNo.AxisName.LCurlingneedleLine].Status.Homed  
AND arrAxisCtrl[AxiseNo.AxisName.SCurlingneedleLine].Status.fActPos <=arrAxisPar[AxiseNo.AxisName.SCurlingneedleLine] .arrTargetPoint[1]+1 
AND arrAxisCtrl[AxiseNo.AxisName.SCurlingneedleLine].Status.Homed 
AND arrCyCtrl[arrCyNo.CylinderName.PullGlueModelCy].Status.ONState
OR Mach_Control.WJ_b.AxisConditionEN THEN
	arrAxisCtrl[AxiseNo.AxisName.TailCurlLine].Cmd.GoPoint_Condition[6]:=TRUE;
ELSE
	arrAxisCtrl[AxiseNo.AxisName.TailCurlLine].Cmd.GoPoint_Condition[6]:=FALSE;	
END_IF

IF  Mach_Control.U.WJ_iMode=3 AND arrAxisCtrl[AxiseNo.AxisName.TailCurlLine].Status.Homed 
AND arrAxisCtrl[AxiseNo.AxisName.TailCurlWhirling].Cmd.arrbRealPoint[1] 
AND arrAxisCtrl[AxiseNo.AxisName.TailCurlSEPTAUpDown].Cmd.arrbRealPoint[1]  
AND arrAxisCtrl[AxiseNo.AxisName.LCurlingneedleLine].Status.fActPos<=arrAxisPar[AxiseNo.AxisName.LCurlingneedleLine].arrTargetPoint[1] +1
AND arrAxisCtrl[AxiseNo.AxisName.LCurlingneedleLine].Status.Homed  
AND arrAxisCtrl[AxiseNo.AxisName.SCurlingneedleLine].Status.fActPos <=arrAxisPar[AxiseNo.AxisName.SCurlingneedleLine] .arrTargetPoint[1]+1 
AND arrAxisCtrl[AxiseNo.AxisName.SCurlingneedleLine].Status.Homed 
AND arrAxisCtrl[AxiseNo.AxisName.TailCurlSEPTALine].Cmd.arrbRealPoint[2]
OR Mach_Control.WJ_b.AxisConditionEN THEN
	arrAxisCtrl[AxiseNo.AxisName.TailCurlLine].Cmd.GoPoint_Condition[7]:=TRUE;
ELSE
	arrAxisCtrl[AxiseNo.AxisName.TailCurlLine].Cmd.GoPoint_Condition[7]:=FALSE;	
END_IF

IF  Mach_Control.U.WJ_iMode=3 AND arrAxisCtrl[AxiseNo.AxisName.TailCurlLine].Status.Homed  
AND arrAxisCtrl[AxiseNo.AxisName.TailCurlWhirling].Cmd.arrbRealPoint[1] 
AND arrAxisCtrl[AxiseNo.AxisName.LCurlingneedleLine].Status.fActPos<=arrAxisPar[AxiseNo.AxisName.LCurlingneedleLine].arrTargetPoint[1]+1 
AND arrAxisCtrl[AxiseNo.AxisName.LCurlingneedleLine].Status.Homed  
AND arrAxisCtrl[AxiseNo.AxisName.SCurlingneedleLine].Status.fActPos <=arrAxisPar[AxiseNo.AxisName.SCurlingneedleLine] .arrTargetPoint[1]+1 
AND arrAxisCtrl[AxiseNo.AxisName.SCurlingneedleLine].Status.Homed  THEN
	arrAxisCtrl[AxiseNo.AxisName.TailCurlLine].Cmd.GoPoint_Condition[8]:=TRUE;
ELSE
	arrAxisCtrl[AxiseNo.AxisName.TailCurlLine].Cmd.GoPoint_Condition[8]:=FALSE;	
END_IF

IF  Mach_Control.U.WJ_iMode=3 AND   arrAxisCtrl[AxiseNo.AxisName.TailCurlLine].Status.Homed  
AND  arrAxisCtrl[AxiseNo.AxisName.TailCurlWhirling].Cmd.arrbRealPoint[1] 
AND(arrAxisCtrl[AxiseNo.AxisName.LCurlingneedleLine].Status.fActPos<=arrAxisPar[AxiseNo.AxisName.LCurlingneedleLine].arrTargetPoint[1]+1 
AND arrAxisCtrl[AxiseNo.AxisName.LCurlingneedleLine].Status.Homed  
AND arrAxisCtrl[AxiseNo.AxisName.SCurlingneedleLine].Status.fActPos <=arrAxisPar[AxiseNo.AxisName.SCurlingneedleLine] .arrTargetPoint[1]+1 
AND arrAxisCtrl[AxiseNo.AxisName.SCurlingneedleLine].Status.Homed 
AND arrCyCtrl[arrCyNo.CylinderName.PoleSplintCy_D].Status.OFFState
AND arrAxisCtrl[AxiseNo.AxisName.TailCurlSEPTALine].Cmd.arrbRealPoint[2]
AND arrAxisCtrl[AxiseNo.AxisName.TailCurlSEPTAUpDown].Cmd.arrbRealPoint[1] ) OR Mach_Control.WJ_b.AxisConditionEN THEN
    arrAxisCtrl[AxiseNo.AxisName.TailCurlLine].Cmd.GoPoint_Condition[9]:=TRUE;
ELSE
	arrAxisCtrl[AxiseNo.AxisName.TailCurlLine].Cmd.GoPoint_Condition[9]:=FALSE;	
END_IF

